(* CODESYS project CODESYS-Libraries
   Author: Ernesto Ponce
   Company: EPonce
   DefaultNamespace: SM_Control
   Description: This Library includes all FB, DUTs and Visualization Faceplates to use the State Machine Logic
   DocFormat: reStructuredText
   LanguageModelAttribute: qualified-access-only
   Placeholder: SM:
   Title: SM_Control
   Version: 1.0

Project tree, tasks and I/O mapping:
  libraries: Util, 3.5.19.0 (System); Standard, 3.5.18.0 (System); VisuSymbols, 4.4.0.0 (System); CmpBitmapPool, 3.5.17.0 (System); VisuDialogs, * (System)
  5ce3da45-db07-42e7-a21c-a00fff4ed8f6|Icons\abort_symbol.png
  5ce3da45-db07-42e7-a21c-a00fff4ed8f6|Icons\camera_icon.png
  5ce3da45-db07-42e7-a21c-a00fff4ed8f6|Icons\home_symbol.png
  5ce3da45-db07-42e7-a21c-a00fff4ed8f6|Icons\menu_icon.png
  5ce3da45-db07-42e7-a21c-a00fff4ed8f6|Icons\pause_symbol.png
  5ce3da45-db07-42e7-a21c-a00fff4ed8f6|Icons\permissives_icon.png
  5ce3da45-db07-42e7-a21c-a00fff4ed8f6|Icons\proceed_symbol.png
  5ce3da45-db07-42e7-a21c-a00fff4ed8f6|Icons\retry_symbol.png
  5ce3da45-db07-42e7-a21c-a00fff4ed8f6|Icons\start_symbol.png
  DUT/
    data type ActiveStep
    data type PermIntlkHMI_cfg
    data type PermIntlkHMI
    data type PermIntlkHMI_ocmd
    data type PermIntlkHMI_sts
    data type SM_HMI
    data type SM_HMI_cfg
    data type SM_HMI_ocmd
    data type SM_HMI_sts
  Function Blocks/
    function block Actuator [ST]: Advance, Reset_Faults, Retract
    function block Permissives [LD]
    program POU [LD]
    function block Real_From_Bytes [ST]
    function block StateMachine [LD]
    function block Step [LD]
  text list GlobalTextList
  global variables GVL
  image pool ImagePool
  Visu_Logic/
    program Visu_Logic [LD]
  Visualizations/
    visualisation Button
    visualisation Menu_Button
    visualisation Permissives_faceplate
    visualisation Screen_Navigation
    visualisation SM_faceplate
*)

// DUT/ActiveStep
TYPE ActiveStep  :
STRUCT
  Step : DINT;
  StatusStepFaulted : BOOL;
  PermsHMI : PermIntlkHMI;
END_STRUCT
END_TYPE

// DUT/PermIntlkHMI_cfg
TYPE PermIntlkHMI_cfg :
STRUCT
  Name : STRING;
  Desc : ARRAY [0..15] OF STRING;
END_STRUCT
END_TYPE

// DUT/PermIntlkHMI
TYPE PermIntlkHMI :
STRUCT
  cfg : PermIntlkHMI_cfg;
  ocmd : PermIntlkHMI_ocmd;
  sts : PermIntlkHMI_sts;
END_STRUCT
END_TYPE

// DUT/PermIntlkHMI_ocmd
TYPE PermIntlkHMI_ocmd :
STRUCT
  ForceOK : BOOL;
END_STRUCT
END_TYPE

// DUT/PermIntlkHMI_sts
TYPE PermIntlkHMI_sts :
STRUCT
  OK : BOOL;
  ForceOK : BOOL;
  PermIntlk : INT;
END_STRUCT
END_TYPE

// DUT/SM_HMI
TYPE SM_HMI :
STRUCT
  cfg : SM_HMI_cfg;
  ocmd : SM_HMI_ocmd;
  sts : SM_HMI_sts;
  NextStatePerms : PermIntlkHMI;
  ActiveStepHMI : PermIntlkHMI;
END_STRUCT
END_TYPE

// DUT/SM_HMI_cfg
TYPE SM_HMI_cfg :
STRUCT
  Name : STRING(40);
  HomePerm : PermIntlkHMI_cfg;
  StartPerm : PermIntlkHMI_cfg;
  ProceedPerm : PermIntlkHMI_cfg;
  AutoIntlk : PermIntlkHMI_cfg;
END_STRUCT
END_TYPE

// DUT/SM_HMI_ocmd
TYPE SM_HMI_ocmd :
STRUCT
  Abort : BOOL;
  Home : BOOL;
  Start : BOOL;
  Stop : BOOL;
  Pause : BOOL;
  Proceed : BOOL;
  Retry : BOOL;
  ActiveStatePermBypass : BOOL;
END_STRUCT
END_TYPE

// DUT/SM_HMI_sts
TYPE SM_HMI_sts :
STRUCT
  Automatic : BOOL;
  Manual : BOOL;
  StepMode : BOOL;
  Homing : BOOL;
  Homed : BOOL;
  Running : BOOL;
  Complete : BOOL;
  Stopping : BOOL;
  Stopped : BOOL;
  Aborting : BOOL;
  Aborted : BOOL;
  Pausing : BOOL;
  Paused : BOOL;
  Proceeding : BOOL;
  Faulted : BOOL;
  ChildFaulted : BOOL;
  ReadyToHome : BOOL;
  ReadyToProceed : BOOL;
  ReadyToStart : BOOL;
  AutoStartRequest : BOOL;
  AutoCycleRequest : BOOL;
  Blocked : BOOL;
  Starved : BOOL;
  Mode : DINT;
  Step : DINT;
  NextStep : DINT;
  ReturnNextStep : DINT;
END_STRUCT
END_TYPE

// GVL

VAR_GLOBAL
	// Global Variables for forcing values
	alwaysTrue : BOOL := TRUE;
	alwaysFalse : BOOL := FALSE;
	
	
	// Colors for Visualization
    indicatorRed: DWORD := 16#FF800000;    // Standard red color, fully opaque
    indicatorGreen: DWORD := 16#FF008000;  // Standard green color, fully opaque
    
    // Modern Color Palette for Buttons
    buttonRed: DWORD := 16#FFE57373;       // Rosy Red, opaque
    buttonRedDarker1: DWORD := 16#FFAF4448; // Crimson Red, opaque
    buttonRedDarker2: DWORD := 16#FF7B3034; // Dark Red, opaque
    buttonRedDarkest: DWORD := 16#FF541F21; // Maroon, opaque
    
    buttonGreen: DWORD := 16#FF81C784;     // Light Green, opaque
    buttonGreenDarker1: DWORD := 16#FF519657; // Medium Sea Green, opaque
    buttonGreenDarker2: DWORD := 16#FF346939; // Dark Green, opaque
    buttonGreenDarkest: DWORD := 16#FF234725; // Dark Olive Green, opaque
    
    buttonGrey: DWORD := 16#FFB0BEC5;      // Blue Grey, opaque
    buttonGreyDarker1: DWORD := 16#FF78909C; // Cadet Blue, opaque
    buttonGreyDarker2: DWORD := 16#FF546E7A; // Steel Blue, opaque
    buttonGreyDarkest: DWORD := 16#FF37474F; // Dark Slate Gray, opaque
	
	// Full Pallet Color Declaration
	
	// Green Palette
	GreenP_1: DWORD := 16#FF859191; // Lightest Green
	GreenP_2: DWORD := 16#FF6F8383; // Light Green
	GreenP_3: DWORD := 16#FF587474; // Medium Light Green
	GreenP_4: DWORD := 16#FF426666; // Medium Green
	GreenP_5: DWORD := 16#FF355151; // Medium Dark Green
	GreenP_6: DWORD := 16#FF283C3C; // Dark Green
	GreenP_7: DWORD := 16#FF1C2828; // Darkest Green
	
	// Grey Palette
	BlueP_1: DWORD := 16#FF8198AD; // Lightest Blue
	BlueP_2: DWORD := 16#FF718CA5; // Light Blue
	BlueP_3: DWORD := 16#FF61809D; // Medium Light Blue
	BlueP_4: DWORD := 16#FF517495; // Medium Blue
	BlueP_5: DWORD := 16#FF41617B; // Medium Dark Blue
	BlueP_6: DWORD := 16#FF314F60; // Dark Blue
	BlueP_7: DWORD := 16#FF213C46; // Darkest Blue
	
	// Purple Palette
	PurpleP_1: DWORD := 16#FF888ECC; // Lightest Purple
	PurpleP_2: DWORD := 16#FF8284C4; // Light Purple
	PurpleP_3: DWORD := 16#FF7C7BBC; // Medium Light Purple
	PurpleP_4: DWORD := 16#FF7571B4; // Medium Purple
	PurpleP_5: DWORD := 16#FF6F68AC; // Medium Dark Purple
	PurpleP_6: DWORD := 16#FF685EA4; // Dark Purple
	PurpleP_7: DWORD := 16#FF62549C; // Darkest Purple
	
	// Yellow Palette
	YellowP_1: DWORD := 16#FFCCC68C; // Lightest Yellow
	YellowP_2: DWORD := 16#FFC4BE80; // Light Yellow
	YellowP_3: DWORD := 16#FFBCB675; // Medium Light Yellow
	YellowP_4: DWORD := 16#FFB4AE6A; // Medium Yellow
	YellowP_5: DWORD := 16#FFACA65F; // Medium Dark Yellow
	YellowP_6: DWORD := 16#FFA49E54; // Dark Yellow
	YellowP_7: DWORD := 16#FF9C9648; // Darkest Yellow
	
	// Brown Palette
	BrownP_1: DWORD := 16#FF99836D; // Lightest Brown
	BrownP_2: DWORD := 16#FF8D7761; // Light Brown
	BrownP_3: DWORD := 16#FF816B55; // Medium Light Brown
	BrownP_4: DWORD := 16#FF755F49; // Medium Brown
	BrownP_5: DWORD := 16#FF69533D; // Medium Dark Brown
	BrownP_6: DWORD := 16#FF5D4731; // Dark Brown
	BrownP_7: DWORD := 16#FF513B25; // Darkest Brown
	
	// Darkened Grey UI Palette
	GreyP_1: DWORD := 16#FFB8B8BC;  // Light Grey
	GreyP_2: DWORD := 16#FFA8A8AC;  // Slightly lighter Grey
	GreyP_3: DWORD := 16#FF98989C;  // Medium Light Grey
	GreyP_4: DWORD := 16#FF88888C;  // True Medium Grey
	GreyP_5: DWORD := 16#FF78787C;  // Medium Dark Grey
	GreyP_6: DWORD := 16#FF68686C;  // Darker Grey
	GreyP_7: DWORD := 16#FF58585C;  // Dark Grey
	
	
	// Visualization Colors Using Pallet
	hover_color : DWORD := BlueP_4;
	normal_color : DWORD := BlueP_6;
	click_color : DWORD := BlueP_6;
	mouseDown_color : DWORD := BlueP_3;
	
	led_colorOFF : DWORD := GreenP_6;
	led_colorON : DWORD := GreenP_3;

END_VAR

// Function Blocks/Actuator
FUNCTION_BLOCK Actuator
VAR_INPUT
	EN:BOOL;
    inRetPermissive: Permissives;
    inAdvPermissive: Permissives;
    inAdvFeedback: BOOL;
    inRetFeedback: BOOL;
    cfgAdvTimeout: TIME;
    cfgRetTimeout: TIME;
END_VAR

VAR_OUTPUT
	ENOut:BOOL;
    outAdvance: BOOL;
    outRetract: BOOL;
	stsAdvancing: BOOL;
    stsAdvanced: BOOL;
	stsRetracting: BOOL;
    stsRetracted: BOOL;
    stsFaulted: BOOL;
    stsFaultCode: INT;
END_VAR

VAR_IN_OUT
	HMI: PermIntlkHMI;
END_VAR


VAR
	timeAdvance:TON;
	timeRetract:TON;	
END_VAR

stsAdvanced:=inAdvFeedback;
stsRetracted:=inRetFeedback;

inAdvPermissive(HMI := HMI);
inRetPermissive(HMI := HMI);


(*
Timeout Fault
Faulted Reason Codes:

- stsFaultCode.0 = 1 = Requested to Advance but !PermsOK
- stsFaultCode.1 = 2 = Requested to Retract but !PermsOK
- stsFaultCode.2 = 4 = Interlocks are not OK
- stsFaultCode.3 = 8 = Advance Timeout
- stsFaultCode.4 = 16 = Retract Timeout
*)
	
timeAdvance(IN:= outAdvance, PT:=cfgAdvTimeout);	
	
IF stsAdvancing AND timeAdvance.Q AND  NOT(inAdvFeedback) THEN
	outAdvance := 0;
	outRetract := 0;
	stsRetracting := 0;
	stsAdvancing := 0;
	stsFaulted := 1;
	stsFaultCode := 8;
END_IF

timeRetract(IN:= outRetract, PT:=cfgRetTimeout);

IF stsRetracting AND timeRetract.Q  AND  NOT(inRetFeedback)THEN
	outAdvance := 0;
	outRetract := 0;
	stsRetracting := 0;
	stsAdvancing := 0;
	stsFaulted := 1;
	stsFaultCode := 16;
END_IF

IF outAdvance AND stsAdvanced THEN	
	stsAdvancing := 0;
END_IF

IF outRetract AND stsRetracted THEN	
	stsRetracting := 0;
END_IF

METHOD Advance : BOOL
VAR_INPUT
	pcmdAdvance:BOOL;
	
END_VAR

VAR
	ONS : R_TRIG;
	
	test:BOOL;
END_VAR
// Advance Logic
ONS(clk:=pcmdAdvance);

IF ONS.Q AND NOT(stsretracting OR stsAdvancing) THEN
	
	outRetract := 0;

	
	IF inAdvPermissive.stsOk THEN
		outAdvance := 1;
		stsAdvancing:= 1;		
	ELSE
		outAdvance := 0;
		outRetract := 0;		
		stsFaulted := 1;
		stsFaultCode := 1;
	END_IF
		
	
END_IF
END_METHOD

METHOD Reset_Faults : BOOL
VAR_INPUT
	pcmdResetFaults:BOOL;
	
END_VAR

VAR
	ONS : R_TRIG;
	
	test:BOOL;
END_VAR
ONS(clk:=pcmdResetFaults);

IF ONS.Q THEN
	outAdvance := 0;
	outRetract := 0;
	stsFaulted := 0;
	stsFaultCode := 0;	
END_IF
END_METHOD

METHOD Retract : BOOL
VAR_INPUT
	pcmdRetract:BOOL;
	
END_VAR

VAR
	ONS : R_TRIG;
	
END_VAR
// Retract Logic
ONS(clk:=pcmdRetract);

IF ONS.Q AND NOT(stsretracting OR stsAdvancing)THEN
	
	outAdvance := 0;

	
	IF inAdvPermissive.stsOk THEN
		outRetract := 1;
		stsRetracting := 1;		
	ELSE
		outAdvance := 0;
		outRetract := 0;
		stsFaulted := 1;
		stsFaultCode := 2;
	END_IF
	
	
END_IF
END_METHOD

END_FUNCTION_BLOCK

// Function Blocks/Permissives
FUNCTION_BLOCK Permissives
VAR_INPUT
	EN: BOOL;
	inPermissives: int;
	ocmdForceOk: BOOL;
	
END_VAR
VAR_OUTPUT
	ENOut: BOOL;
	stsOk: BOOL;
	stsForceOk: BOOL;
	
END_VAR
VAR
END_VAR

VAR_IN_OUT
	HMI: PermIntlkHMI;
END_VAR
VAR // added by the converter: edge detectors and wires of the graphical bodies
    _w1, _w2 : BOOL;
END_VAR

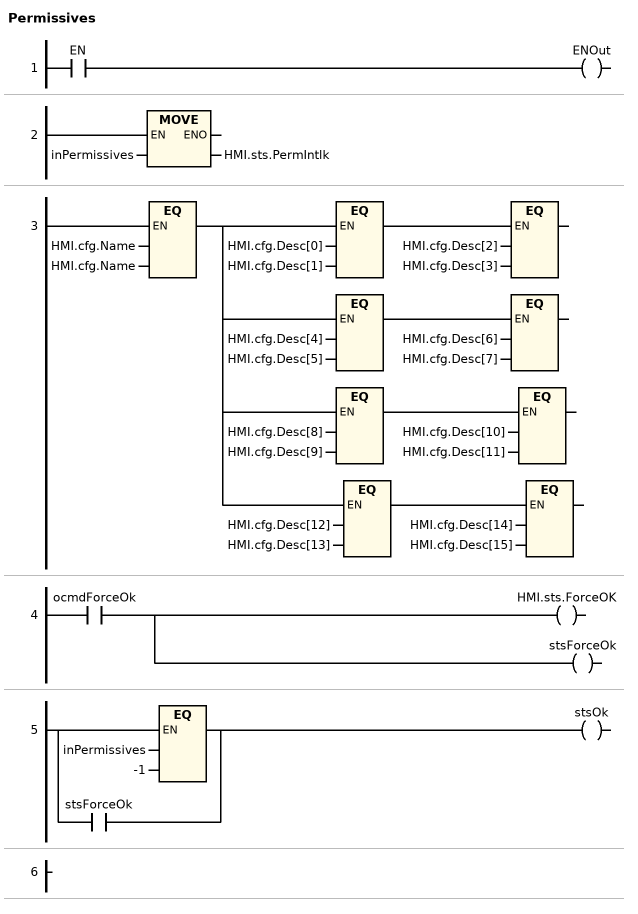
// NETWORK 1
ENOut := EN;

// NETWORK 2
HMI.sts.PermIntlk := inPermissives;

// NETWORK 3
_w1 := HMI.cfg.Name = HMI.cfg.Name;
(* _w1 AND HMI.cfg.Desc[0] = HMI.cfg.Desc[1] AND HMI.cfg.Desc[2] = HMI.cfg.Desc[3]; result not used *)
(* _w1 AND HMI.cfg.Desc[4] = HMI.cfg.Desc[5] AND HMI.cfg.Desc[6] = HMI.cfg.Desc[7]; result not used *)
(* _w1 AND HMI.cfg.Desc[8] = HMI.cfg.Desc[9] AND HMI.cfg.Desc[10] = HMI.cfg.Desc[11]; result not used *)
(* _w1 AND HMI.cfg.Desc[12] = HMI.cfg.Desc[13] AND HMI.cfg.Desc[14] = HMI.cfg.Desc[15]; result not used *)

// NETWORK 4
HMI.sts.ForceOK := ocmdForceOk;
stsForceOk := ocmdForceOk;

// NETWORK 5
_w2 := stsForceOk;
IF NOT _w2 THEN
    _w2 := inPermissives = -1;
END_IF
stsOk := _w2;

// NETWORK 6

END_FUNCTION_BLOCK

// Function Blocks/POU
PROGRAM POU
VAR
	
END_VAR

// NETWORK 1

END_PROGRAM

// Function Blocks/Real_From_Bytes
FUNCTION_BLOCK Real_From_Bytes
VAR_INPUT
    Byte1: BYTE; 
    Byte2: BYTE; 
    Byte3: BYTE; 
    Byte4: BYTE; 
END_VAR

VAR_OUTPUT
    RealValue: REAL; // The resulting REAL value
    
END_VAR

VAR
    Word1: WORD;
    Word2: WORD;
    Word3: WORD;
    Word4: WORD;
    Dword1: DWORD;
    Dword2: DWORD;
    Dword3: DWORD;
    Dword4: DWORD;
    ShiftedDword2: DWORD;
    ShiftedDword3: DWORD;
    ShiftedDword4: DWORD;
	CombinedDword: DWORD;
    ptrRealValue: POINTER TO REAL;
END_VAR

 // Convert each byte to a WORD
    Word1 := BYTE_TO_WORD(Byte4);
    Word2 := BYTE_TO_WORD(Byte1);
    Word3 := BYTE_TO_WORD(Byte2);
    Word4 := BYTE_TO_WORD(Byte3);

    // Convert each WORD to a DWORD
    Dword1 := WORD_TO_DWORD(Word1);
    Dword2 := WORD_TO_DWORD(Word2);
    Dword3 := WORD_TO_DWORD(Word3);
    Dword4 := WORD_TO_DWORD(Word4);

    // Shift DWORDs to the correct position
    ShiftedDword2 := SHL(Dword2, 8);
    ShiftedDword3 := SHL(Dword3, 16);
    ShiftedDword4 := SHL(Dword4, 24);

    // Combine the DWORDs into one DWORD assuming big-endian order
    CombinedDword := Dword1 OR ShiftedDword2 OR ShiftedDword3 OR ShiftedDword4;

    // Use pointer method to convert the combined DWORD to REAL
    ptrRealValue := ADR(CombinedDword);
    RealValue := ptrRealValue^;

END_FUNCTION_BLOCK

// Function Blocks/StateMachine
FUNCTION_BLOCK StateMachine

VAR_INPUT
    EnableIn: BOOL;
    cfgAutoRun: BOOL;
    inpAutoIntlk: INT:= -1;
    inpBlockedCondition: DINT;
    inpHomePerm: INT := -1;
    inpProceedPerm: INT := -1;
    inpStartPerm: INT := -1;
    inpStarvedCondition: DINT;
    inpSubmoduleFaulted: BOOL;
    NextStep: DINT;
    pcmdAbort: BOOL;
    pcmdCompleteState: BOOL;
    pcmdHome: BOOL;
    pcmdPause: BOOL;
    pcmdProceed: BOOL;
    pcmdRetry: BOOL;
    pcmdStart: BOOL;
    pcmdStop: BOOL;
END_VAR

VAR_OUTPUT
    EnableOut: BOOL;
    outRetry: BOOL;
    stsAborted: BOOL;
    stsAborting: BOOL;
    stsActiveState: BOOL;
    stsAutoCycleRequest: BOOL;
    stsAutoIntlkOK: BOOL;
    stsAutomatic: BOOL;
    stsAutoStartRequest: BOOL;
    stsBlocked: BOOL;
    stsBlockedCondition: DINT;
    stsComplete: BOOL;
    stsFaulted: BOOL;
    stsHomed: BOOL;
    stsHomePermOk: BOOL;
    stsHoming: BOOL;
    stsManual: BOOL;
    stsMode: DINT;
    stsPaused: BOOL;
    stsPausing: BOOL;
    stsProceeding: BOOL;
    stsProceedPermOK: BOOL;
    stsReadyToHome: BOOL;
    stsReadyToProceed: BOOL;
    stsReadyToStart: BOOL;
    stsReturnNextStep: DINT;
    stsRunning: BOOL;
    stsStartPermOK: BOOL;
    stsStarved: BOOL;
    stsStarvedCondition: DINT;
    stsStep: DINT;
    stsStepTimerSeconds: REAL;
    stsStopped: BOOL;
    stsStopping: BOOL;
    stsSubmoduleFaulted: BOOL;
    stsWaitingState: BOOL;
	stsState: INT;
	stsStateString: STRING;
	stsReturnState: INT;
	stsLastState: INT;
END_VAR


VAR CONSTANT 
	internalClearStep: ActiveStep;  
	EmptyHMIPerm: PermIntlkHMI;
	
	// All internal steps
	internalStateRunning: INT := 1;
    internalStateStopping: INT := 2;
    internalStateHoming: INT := 4;
    internalStateAborting: INT := 8;
    internalStateHomed: INT := 16;
    internalStateStopped: INT := 32;
    internalStateAborted: INT := 64;
    internalStateComplete: INT := 128;
    internalStatePausing: INT := 256;
    internalStatePaused: INT := 512;
    internalStateProceeding: INT := 1024;
END_VAR

VAR
    AbortRequested: BOOL;
    AutoStartRequested: BOOL;
    CompleteStateRequested: BOOL;
    HomeRequested: BOOL;
    PauseRequested: BOOL;
    ProceedRequested: BOOL;
    RetryComplete: BOOL;
    RetryRequested: BOOL;
    StartRequested: BOOL;
    StopRequested: BOOL;
    StepTimer: TON;

    internalLsOdd: DINT;
   	internalONS: DINT;
 	R_TRIG_0: R_TRIG;
	R_TRIG_1: R_TRIG;
	R_TRIG_2: R_TRIG;
	R_TRIG_3: R_TRIG;
	internalTimerReset: BOOL;
	
	internalPauseStep: ActiveStep;
    internalPreviousState: INT;
	internalAutoIntlk: Permissives;
    internalAutoIntlk_HMI: PermIntlkHMI;
    internalProceedPerm: Permissives;
    internalProceedPerm_HMI: PermIntlkHMI;
    internalStartPerm: Permissives;
    internalStartPerm_HMI: PermIntlkHMI;
	internalHomePerm: Permissives;
    internalHomePerm_HMI: PermIntlkHMI;
	internalStepHistoryMax: DINT;
END_VAR


VAR_IN_OUT 
    HMI: SM_HMI;
    CurrentStep: ActiveStep;
    
END_VAR
VAR // added by the converter: edge detectors and wires of the graphical bodies
    _w1, _w2, _w3, _w4, _w5, _w6, _w7, _w8, _w9, _w10, _w11, _w12, _w13, _w14, _w15, _w16, _w17, _w18, _w19, _w20, _w21, _w22, _w23, _w24, _w25, _w26, _w27, _w28, _w29, _w30, _w31, _w32, _w33, _w34, _w35, _w36, _w37, _w38, _w39, _w40, _w41, _w42, _w43, _w44 : BOOL;
    _rt1, _rt2 : R_TRIG;
END_VAR

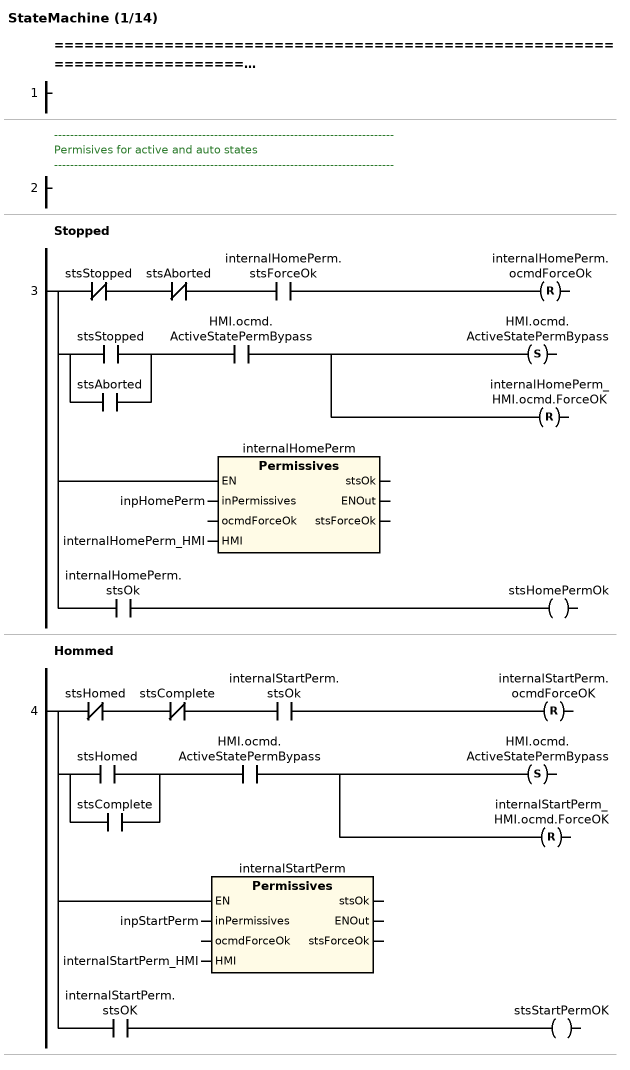
// NETWORK 1: ============================================================================ State Machine ============================================================================ (disabled)

// NETWORK 2
// -------------------------------------------------------------------------------------
//
// Permisives for active and auto states
//
// -------------------------------------------------------------------------------------

// NETWORK 3: Stopped
internalHomePerm.ocmdForceOk R= NOT stsStopped AND NOT stsAborted AND internalHomePerm.stsForceOk;
_w1 := (stsStopped OR stsAborted) AND HMI.ocmd.ActiveStatePermBypass;
HMI.ocmd.ActiveStatePermBypass S= _w1;
internalHomePerm_HMI.ocmd.ForceOK R= _w1;
internalHomePerm(EN := TRUE, inPermissives := inpHomePerm, HMI := internalHomePerm_HMI); // Permissives
stsHomePermOk := internalHomePerm.stsOk;

// NETWORK 4: Hommed
internalStartPerm.ocmdForceOK R= NOT stsHomed AND NOT stsComplete AND internalStartPerm.stsOk;
_w2 := (stsHomed OR stsComplete) AND HMI.ocmd.ActiveStatePermBypass;
HMI.ocmd.ActiveStatePermBypass S= _w2;
internalStartPerm_HMI.ocmd.ForceOK R= _w2;
internalStartPerm(EN := TRUE, inPermissives := inpStartPerm, HMI := internalStartPerm_HMI); // Permissives
stsStartPermOK := internalStartPerm.stsOK;

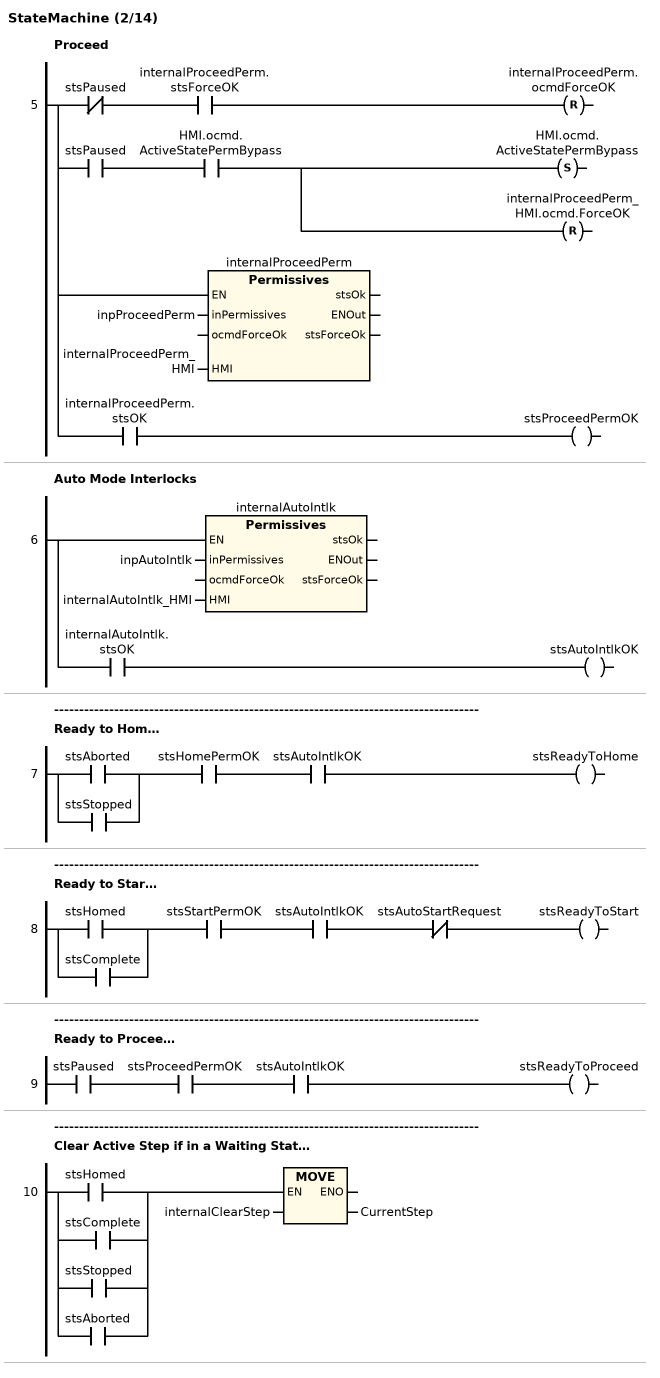
// NETWORK 5: Proceed
internalProceedPerm.ocmdForceOK R= NOT stsPaused AND internalProceedPerm.stsForceOK;
_w3 := stsPaused AND HMI.ocmd.ActiveStatePermBypass;
HMI.ocmd.ActiveStatePermBypass S= _w3;
internalProceedPerm_HMI.ocmd.ForceOK R= _w3;
internalProceedPerm(EN := TRUE, inPermissives := inpProceedPerm, HMI := internalProceedPerm_HMI); // Permissives
stsProceedPermOK := internalProceedPerm.stsOK;

// NETWORK 6: Auto Mode Interlocks
internalAutoIntlk(EN := TRUE, inPermissives := inpAutoIntlk, HMI := internalAutoIntlk_HMI); // Permissives
stsAutoIntlkOK := internalAutoIntlk.stsOK;

// NETWORK 7: ------------------------------------------------------------------------------------- Ready to Home - if stopped or aborted - if Perms are OK -------------------------------------------------------------------------------------
stsReadyToHome := (stsAborted OR stsStopped) AND stsHomePermOK AND stsAutoIntlkOK;

// NETWORK 8: ------------------------------------------------------------------------------------- Ready to Start - if homed or complete - if Perms are OK -------------------------------------------------------------------------------------
stsReadyToStart := (stsHomed OR stsComplete) AND stsStartPermOK AND stsAutoIntlkOK AND NOT stsAutoStartRequest;

// NETWORK 9: ------------------------------------------------------------------------------------- Ready to Proceed - if paused - if Perms are OK -------------------------------------------------------------------------------------
stsReadyToProceed := stsPaused AND stsProceedPermOK AND stsAutoIntlkOK;

// NETWORK 10: ------------------------------------------------------------------------------------- Clear Active Step if in a Waiting State -------------------------------------------------------------------------------------
IF stsHomed OR stsComplete OR stsStopped OR stsAborted THEN CurrentStep := internalClearStep; END_IF

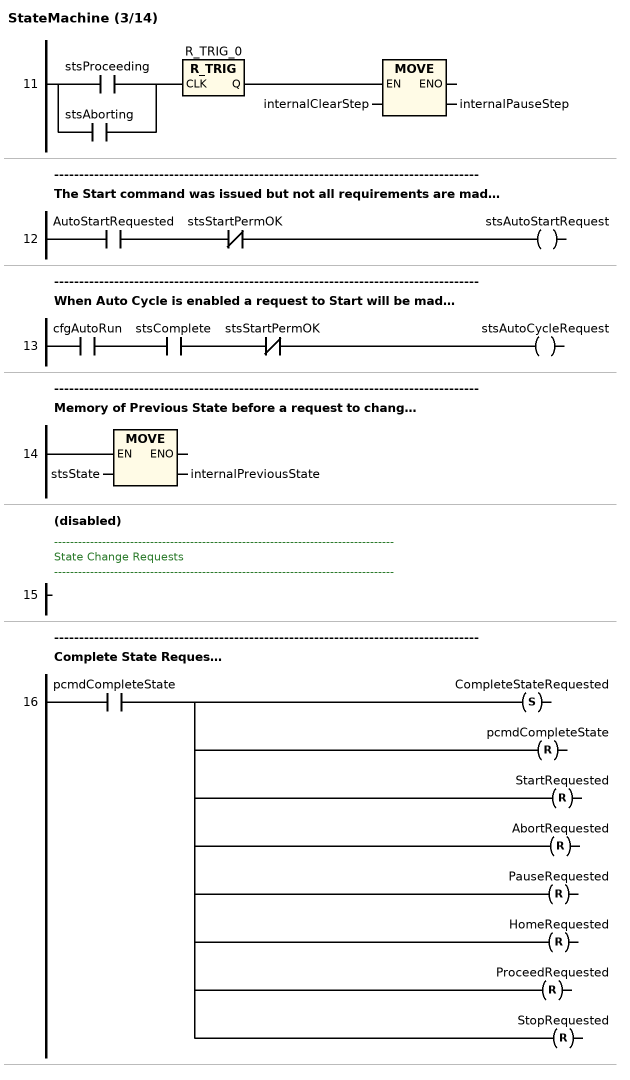
// NETWORK 11
R_TRIG_0(CLK := stsProceeding OR stsAborting); // R_TRIG
IF R_TRIG_0.Q THEN internalPauseStep := internalClearStep; END_IF

// NETWORK 12: ------------------------------------------------------------------------------------- The Start command was issued but not all requirements are made The request will be remembered and this will happen as soon as everything is ready to Start -------------------------------------------------------------------------------------
stsAutoStartRequest := AutoStartRequested AND NOT stsStartPermOK;

// NETWORK 13: ------------------------------------------------------------------------------------- When Auto Cycle is enabled a request to Start will be made as soon as the previous cycle is Complete -------------------------------------------------------------------------------------
stsAutoCycleRequest := cfgAutoRun AND stsComplete AND NOT stsStartPermOK;

// NETWORK 14: ------------------------------------------------------------------------------------- Memory of Previous State before a request to change -------------------------------------------------------------------------------------
internalPreviousState := stsState;

// NETWORK 15 (disabled)
// -------------------------------------------------------------------------------------
//
// State Change Requests
//
// -------------------------------------------------------------------------------------

// NETWORK 16: ------------------------------------------------------------------------------------- Complete State Request -------------------------------------------------------------------------------------
_w4 := pcmdCompleteState;
CompleteStateRequested S= _w4;
pcmdCompleteState R= _w4;
StartRequested R= _w4;
AbortRequested R= _w4;
PauseRequested R= _w4;
HomeRequested R= _w4;
ProceedRequested R= _w4;
StopRequested R= _w4;

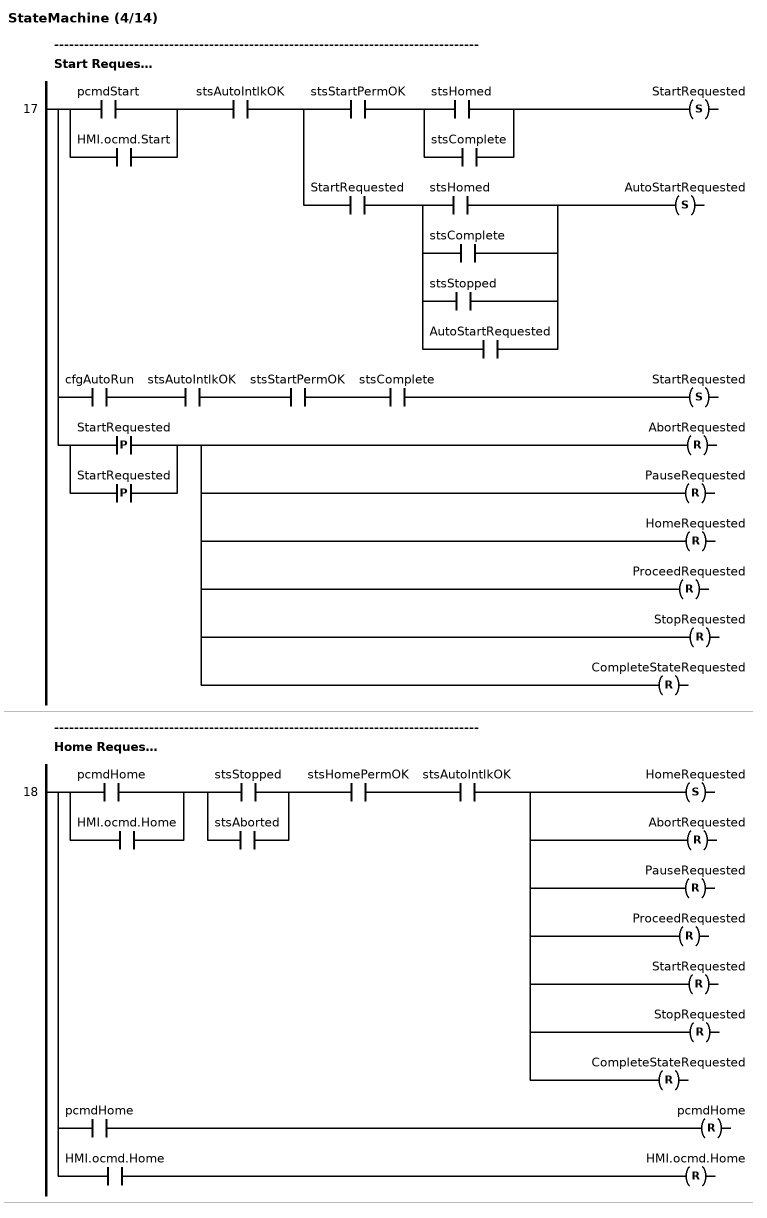
// NETWORK 17: ------------------------------------------------------------------------------------- Start Request -------------------------------------------------------------------------------------
_w5 := (pcmdStart OR HMI.ocmd.Start) AND stsAutoIntlkOK;
StartRequested S= _w5 AND stsStartPermOK AND (stsHomed OR stsComplete);
AutoStartRequested S= _w5 AND StartRequested AND (stsHomed OR stsComplete OR stsStopped OR AutoStartRequested);
StartRequested S= cfgAutoRun AND stsAutoIntlkOK AND stsStartPermOK AND stsComplete;
_rt1(CLK := StartRequested);
_rt2(CLK := StartRequested);
_w6 := _rt1.Q OR _rt2.Q;
AbortRequested R= _w6;
PauseRequested R= _w6;
HomeRequested R= _w6;
ProceedRequested R= _w6;
StopRequested R= _w6;
CompleteStateRequested R= _w6;

// NETWORK 18: ------------------------------------------------------------------------------------- Home Request -------------------------------------------------------------------------------------
_w7 := (pcmdHome OR HMI.ocmd.Home) AND (stsStopped OR stsAborted) AND stsHomePermOK AND stsAutoIntlkOK;
HomeRequested S= _w7;
AbortRequested R= _w7;
PauseRequested R= _w7;
ProceedRequested R= _w7;
StartRequested R= _w7;
StopRequested R= _w7;
CompleteStateRequested R= _w7;
pcmdHome R= pcmdHome;
HMI.ocmd.Home R= HMI.ocmd.Home;

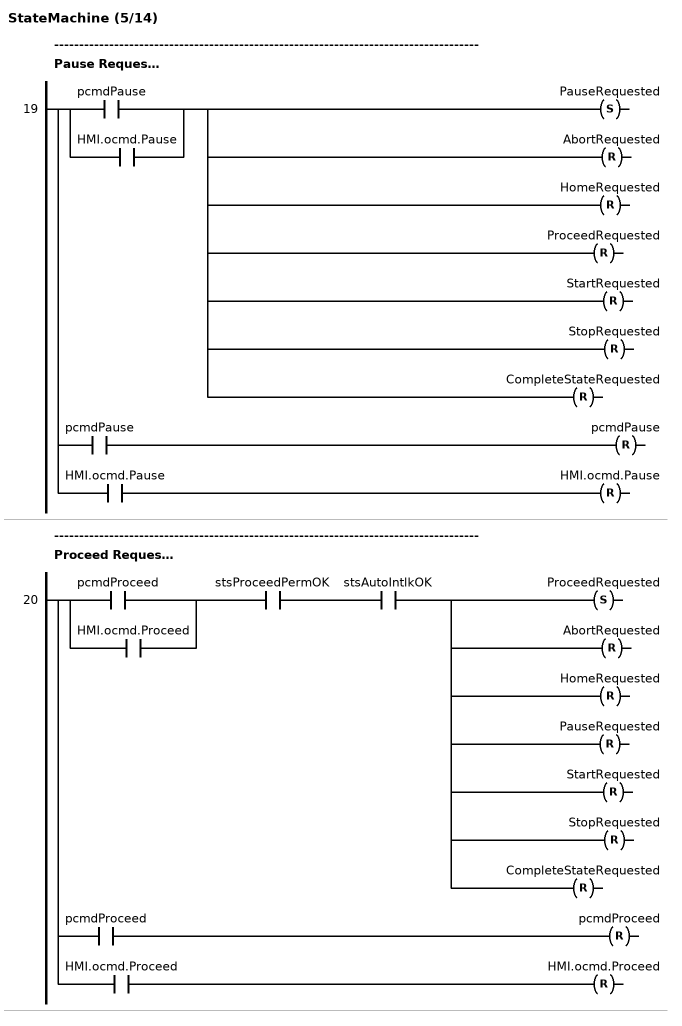
// NETWORK 19: ------------------------------------------------------------------------------------- Pause Request -------------------------------------------------------------------------------------
_w8 := pcmdPause OR HMI.ocmd.Pause;
PauseRequested S= _w8;
AbortRequested R= _w8;
HomeRequested R= _w8;
ProceedRequested R= _w8;
StartRequested R= _w8;
StopRequested R= _w8;
CompleteStateRequested R= _w8;
pcmdPause R= pcmdPause;
HMI.ocmd.Pause R= HMI.ocmd.Pause;

// NETWORK 20: ------------------------------------------------------------------------------------- Proceed Request -------------------------------------------------------------------------------------
_w9 := (pcmdProceed OR HMI.ocmd.Proceed) AND stsProceedPermOK AND stsAutoIntlkOK;
ProceedRequested S= _w9;
AbortRequested R= _w9;
HomeRequested R= _w9;
PauseRequested R= _w9;
StartRequested R= _w9;
StopRequested R= _w9;
CompleteStateRequested R= _w9;
pcmdProceed R= pcmdProceed;
HMI.ocmd.Proceed R= HMI.ocmd.Proceed;

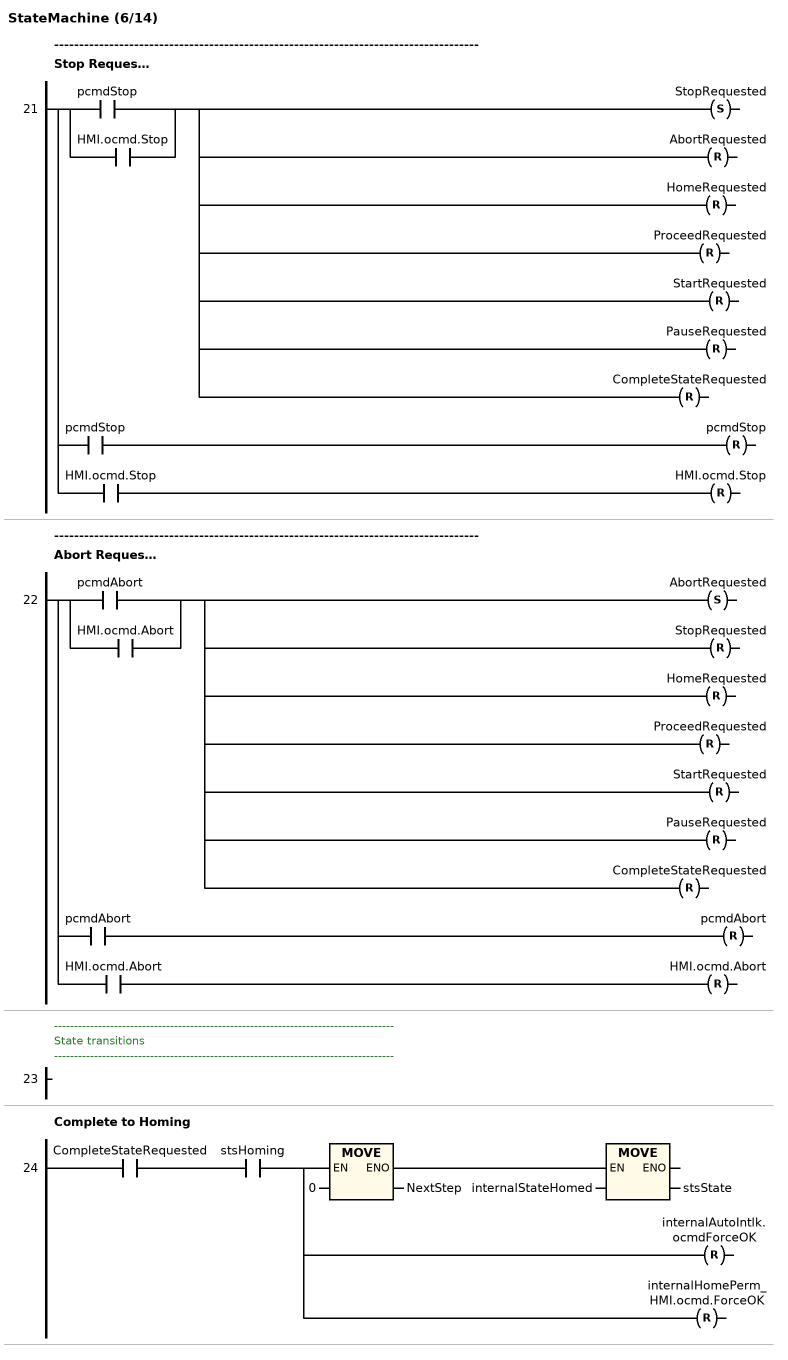
// NETWORK 21: ------------------------------------------------------------------------------------- Stop Request -------------------------------------------------------------------------------------
_w10 := pcmdStop OR HMI.ocmd.Stop;
StopRequested S= _w10;
AbortRequested R= _w10;
HomeRequested R= _w10;
ProceedRequested R= _w10;
StartRequested R= _w10;
PauseRequested R= _w10;
CompleteStateRequested R= _w10;
pcmdStop R= pcmdStop;
HMI.ocmd.Stop R= HMI.ocmd.Stop;

// NETWORK 22: ------------------------------------------------------------------------------------- Abort Request -------------------------------------------------------------------------------------
_w11 := pcmdAbort OR HMI.ocmd.Abort;
AbortRequested S= _w11;
StopRequested R= _w11;
HomeRequested R= _w11;
ProceedRequested R= _w11;
StartRequested R= _w11;
PauseRequested R= _w11;
CompleteStateRequested R= _w11;
pcmdAbort R= pcmdAbort;
HMI.ocmd.Abort R= HMI.ocmd.Abort;

// NETWORK 23
// -------------------------------------------------------------------------------------
//
// State transitions
//
// -------------------------------------------------------------------------------------

// NETWORK 24: Complete to Homing
_w12 := CompleteStateRequested AND stsHoming;
IF _w12 THEN NextStep := 0; END_IF
IF _w12 THEN stsState := internalStateHomed; END_IF
internalAutoIntlk.ocmdForceOK R= _w12;
internalHomePerm_HMI.ocmd.ForceOK R= _w12;

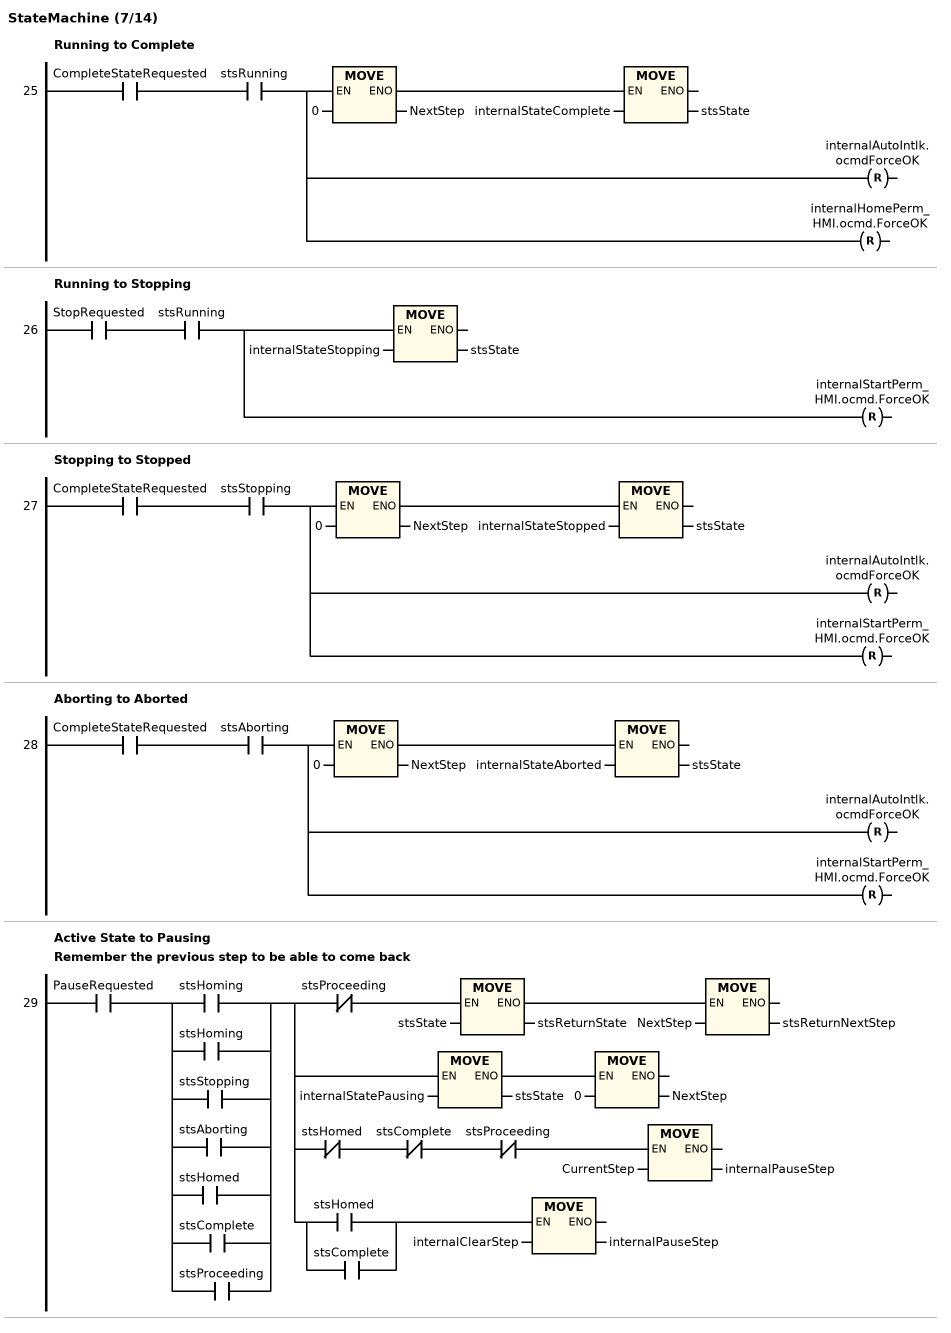
// NETWORK 25: Running to Complete
_w13 := CompleteStateRequested AND stsRunning;
IF _w13 THEN NextStep := 0; END_IF
IF _w13 THEN stsState := internalStateComplete; END_IF
internalAutoIntlk.ocmdForceOK R= _w13;
internalHomePerm_HMI.ocmd.ForceOK R= _w13;

// NETWORK 26: Running to Stopping
_w14 := StopRequested AND stsRunning;
IF _w14 THEN stsState := internalStateStopping; END_IF
internalStartPerm_HMI.ocmd.ForceOK R= _w14;

// NETWORK 27: Stopping to Stopped
_w15 := CompleteStateRequested AND stsStopping;
IF _w15 THEN NextStep := 0; END_IF
IF _w15 THEN stsState := internalStateStopped; END_IF
internalAutoIntlk.ocmdForceOK R= _w15;
internalStartPerm_HMI.ocmd.ForceOK R= _w15;

// NETWORK 28: Aborting to Aborted
_w16 := CompleteStateRequested AND stsAborting;
IF _w16 THEN NextStep := 0; END_IF
IF _w16 THEN stsState := internalStateAborted; END_IF
internalAutoIntlk.ocmdForceOK R= _w16;
internalStartPerm_HMI.ocmd.ForceOK R= _w16;

// NETWORK 29: Active State to Pausing Remember the previous step to be able to come back
_w17 := PauseRequested AND (stsHoming OR stsHoming OR stsStopping OR stsAborting OR stsHomed OR stsComplete OR stsProceeding);
IF _w17 AND NOT stsProceeding THEN stsReturnState := stsState; END_IF
IF _w17 AND NOT stsProceeding THEN stsReturnNextStep := NextStep; END_IF
IF _w17 THEN stsState := internalStatePausing; END_IF
IF _w17 THEN NextStep := 0; END_IF
IF _w17 AND NOT stsHomed AND NOT stsComplete AND NOT stsProceeding THEN internalPauseStep := CurrentStep; END_IF
IF _w17 AND (stsHomed OR stsComplete) THEN internalPauseStep := internalClearStep; END_IF

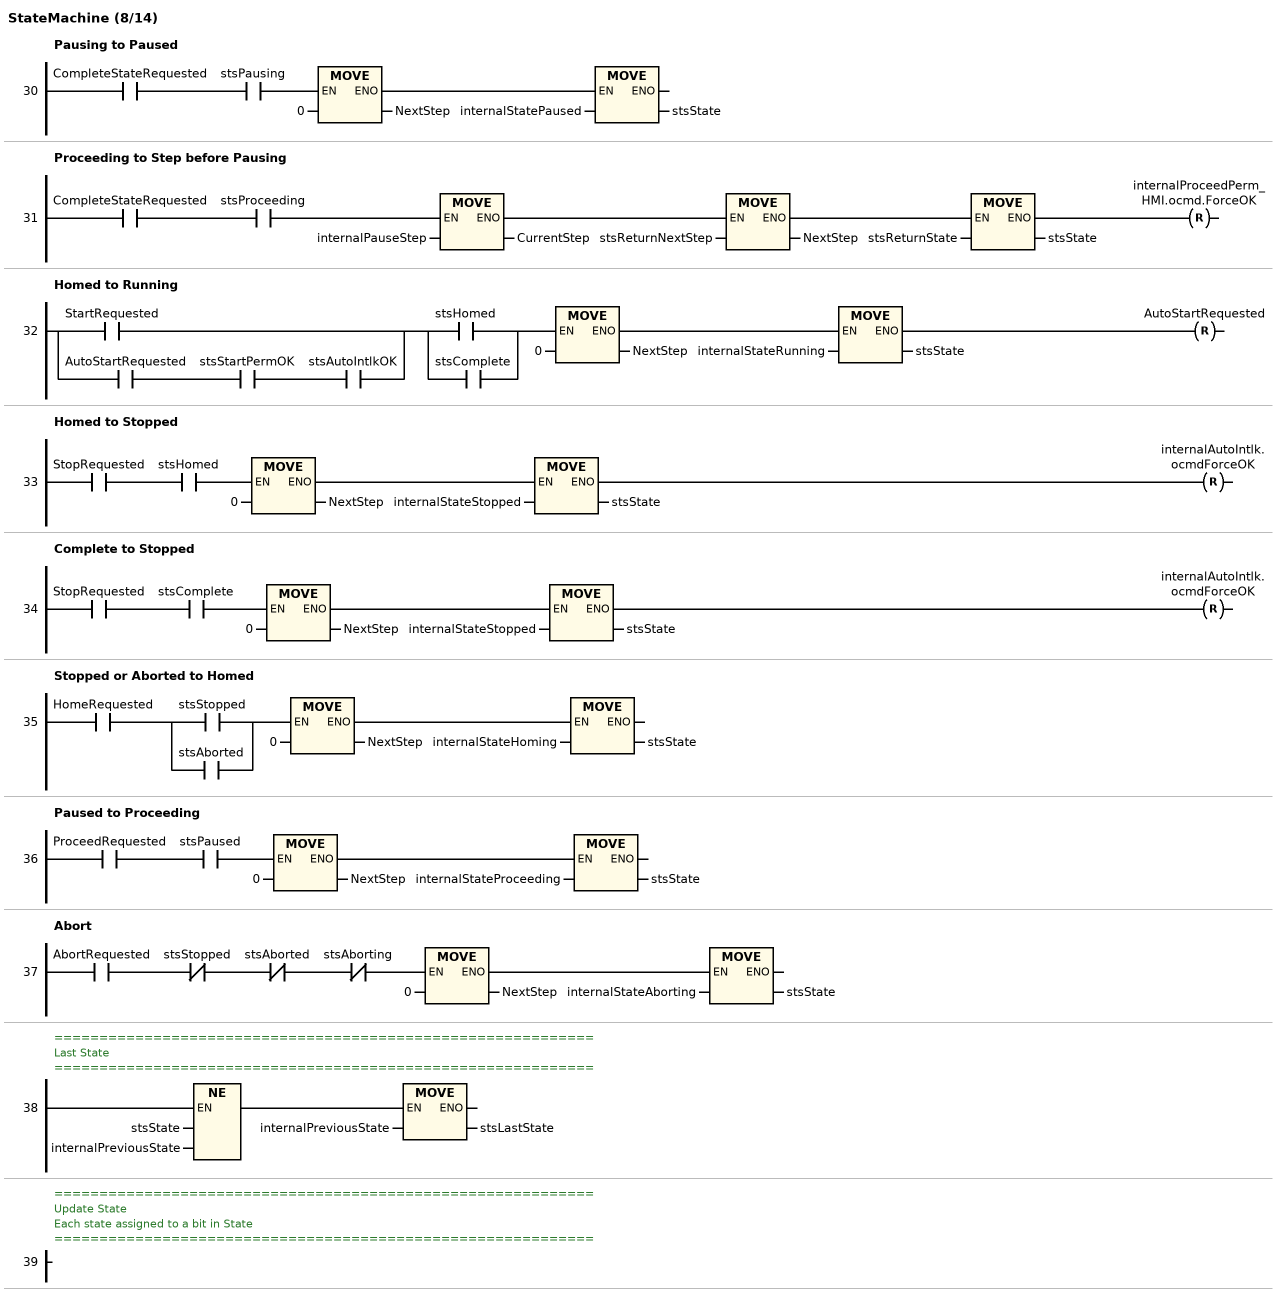
// NETWORK 30: Pausing to Paused
_w18 := CompleteStateRequested AND stsPausing;
IF _w18 THEN NextStep := 0; END_IF
IF _w18 THEN stsState := internalStatePaused; END_IF

// NETWORK 31: Proceeding to Step before Pausing
_w19 := CompleteStateRequested AND stsProceeding;
IF _w19 THEN CurrentStep := internalPauseStep; END_IF
IF _w19 THEN NextStep := stsReturnNextStep; END_IF
IF _w19 THEN stsState := stsReturnState; END_IF
internalProceedPerm_HMI.ocmd.ForceOK R= _w19;

// NETWORK 32: Homed to Running
_w20 := (StartRequested OR AutoStartRequested AND stsStartPermOK AND stsAutoIntlkOK) AND (stsHomed OR stsComplete);
IF _w20 THEN NextStep := 0; END_IF
IF _w20 THEN stsState := internalStateRunning; END_IF
AutoStartRequested R= _w20;

// NETWORK 33: Homed to Stopped
_w21 := StopRequested AND stsHomed;
IF _w21 THEN NextStep := 0; END_IF
IF _w21 THEN stsState := internalStateStopped; END_IF
internalAutoIntlk.ocmdForceOK R= _w21;

// NETWORK 34: Complete to Stopped
_w22 := StopRequested AND stsComplete;
IF _w22 THEN NextStep := 0; END_IF
IF _w22 THEN stsState := internalStateStopped; END_IF
internalAutoIntlk.ocmdForceOK R= _w22;

// NETWORK 35: Stopped or Aborted to Homed
_w23 := HomeRequested AND (stsStopped OR stsAborted);
IF _w23 THEN NextStep := 0; END_IF
IF _w23 THEN stsState := internalStateHoming; END_IF

// NETWORK 36: Paused to Proceeding
_w24 := ProceedRequested AND stsPaused;
IF _w24 THEN NextStep := 0; END_IF
IF _w24 THEN stsState := internalStateProceeding; END_IF

// NETWORK 37: Abort
_w25 := AbortRequested AND NOT stsStopped AND NOT stsAborted AND NOT stsAborting;
IF _w25 THEN NextStep := 0; END_IF
IF _w25 THEN stsState := internalStateAborting; END_IF

// NETWORK 38
// ============================================================
// Last State
// ============================================================
IF stsState <> internalPreviousState THEN stsLastState := internalPreviousState; END_IF

// NETWORK 39
// ============================================================
// Update State
// Each state assigned to a bit in State
// ============================================================

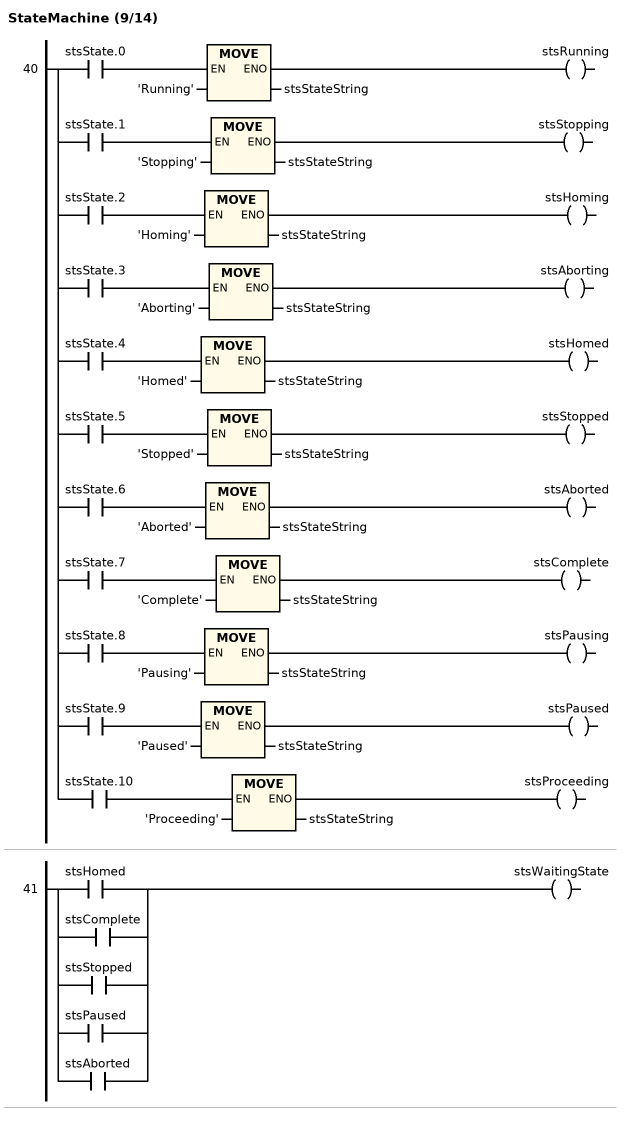
// NETWORK 40
_w26 := stsState.0;
IF _w26 THEN stsStateString := 'Running'; END_IF
stsRunning := _w26;
_w27 := stsState.1;
IF _w27 THEN stsStateString := 'Stopping'; END_IF
stsStopping := _w27;
_w28 := stsState.2;
IF _w28 THEN stsStateString := 'Homing'; END_IF
stsHoming := _w28;
_w29 := stsState.3;
IF _w29 THEN stsStateString := 'Aborting'; END_IF
stsAborting := _w29;
_w30 := stsState.4;
IF _w30 THEN stsStateString := 'Homed'; END_IF
stsHomed := _w30;
_w31 := stsState.5;
IF _w31 THEN stsStateString := 'Stopped'; END_IF
stsStopped := _w31;
_w32 := stsState.6;
IF _w32 THEN stsStateString := 'Aborted'; END_IF
stsAborted := _w32;
_w33 := stsState.7;
IF _w33 THEN stsStateString := 'Complete'; END_IF
stsComplete := _w33;
_w34 := stsState.8;
IF _w34 THEN stsStateString := 'Pausing'; END_IF
stsPausing := _w34;
_w35 := stsState.9;
IF _w35 THEN stsStateString := 'Paused'; END_IF
stsPaused := _w35;
_w36 := stsState.10;
IF _w36 THEN stsStateString := 'Proceeding'; END_IF
stsProceeding := _w36;

// NETWORK 41
stsWaitingState := stsHomed OR stsComplete OR stsStopped OR stsPaused OR stsAborted;

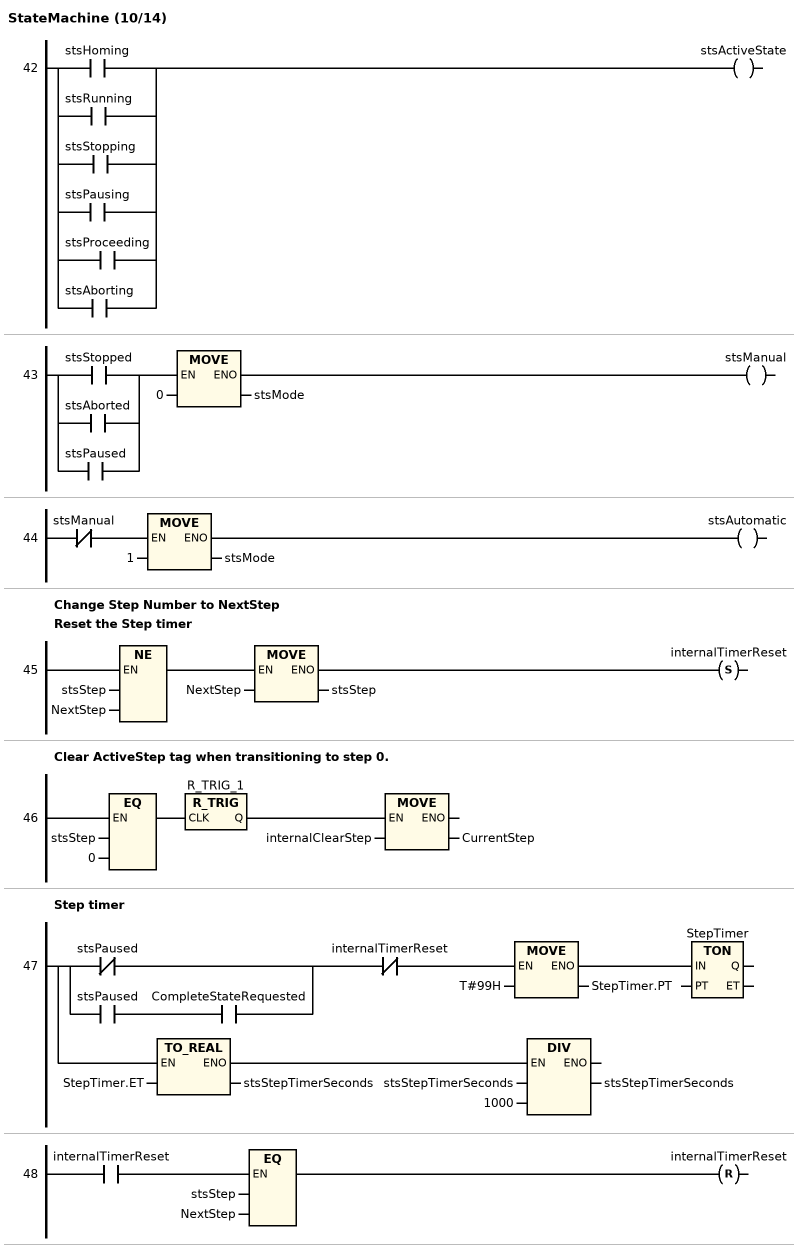
// NETWORK 42
stsActiveState := stsHoming OR stsRunning OR stsStopping OR stsPausing OR stsProceeding OR stsAborting;

// NETWORK 43
_w37 := stsStopped OR stsAborted OR stsPaused;
IF _w37 THEN stsMode := 0; END_IF
stsManual := _w37;

// NETWORK 44
_w38 := NOT stsManual;
IF _w38 THEN stsMode := 1; END_IF
stsAutomatic := _w38;

// NETWORK 45: Change Step Number to NextStep Reset the Step timer
_w39 := stsStep <> NextStep;
IF _w39 THEN stsStep := NextStep; END_IF
internalTimerReset S= _w39;

// NETWORK 46: Clear ActiveStep tag when transitioning to step 0.
R_TRIG_1(CLK := stsStep = 0); // R_TRIG
IF R_TRIG_1.Q THEN CurrentStep := internalClearStep; END_IF

// NETWORK 47: Step timer
_w40 := (NOT stsPaused OR stsPaused AND CompleteStateRequested) AND NOT internalTimerReset;
IF _w40 THEN StepTimer.PT := T#99H; END_IF
StepTimer(IN := _w40); // TON
stsStepTimerSeconds := TO_REAL(StepTimer.ET);
stsStepTimerSeconds := stsStepTimerSeconds / 1000;

// NETWORK 48
internalTimerReset R= internalTimerReset AND stsStep = NextStep;

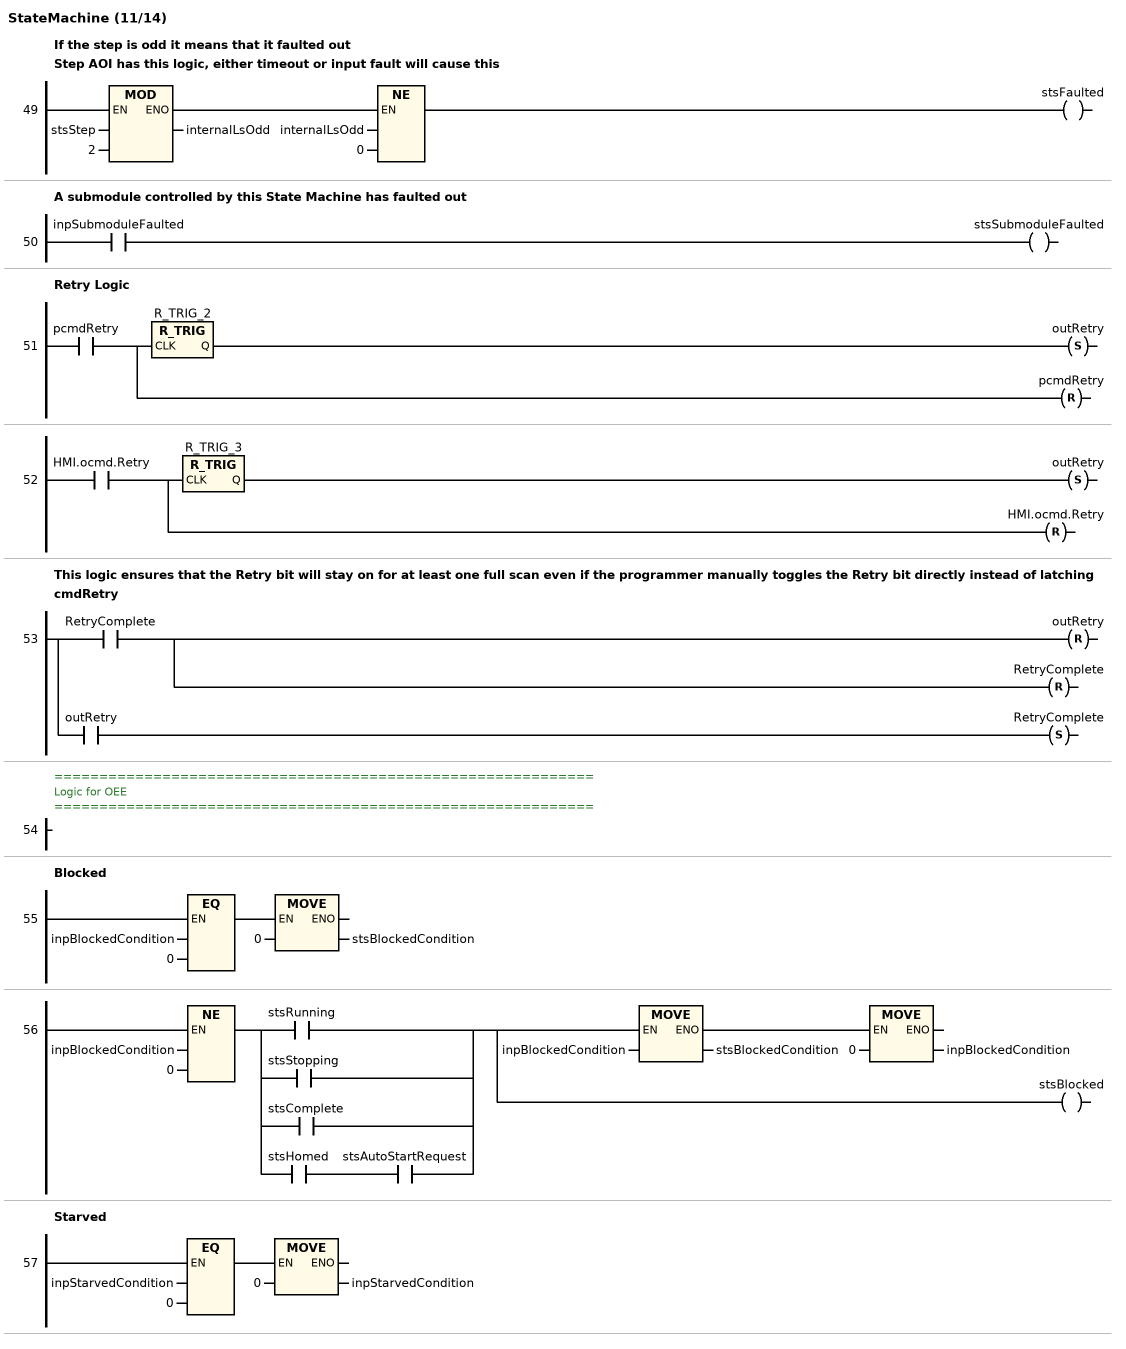
// NETWORK 49: If the step is odd it means that it faulted out Step AOI has this logic, either timeout or input fault will cause this
internalLsOdd := stsStep MOD 2;
stsFaulted := internalLsOdd <> 0;

// NETWORK 50: A submodule controlled by this State Machine has faulted out
stsSubmoduleFaulted := inpSubmoduleFaulted;

// NETWORK 51: Retry Logic
_w41 := pcmdRetry;
R_TRIG_2(CLK := _w41); // R_TRIG
outRetry S= R_TRIG_2.Q;
pcmdRetry R= _w41;

// NETWORK 52
_w42 := HMI.ocmd.Retry;
R_TRIG_3(CLK := _w42); // R_TRIG
outRetry S= R_TRIG_3.Q;
HMI.ocmd.Retry R= _w42;

// NETWORK 53: This logic ensures that the Retry bit will stay on for at least one full scan even if the programmer manually toggles the Retry bit directly instead of latching cmdRetry
outRetry R= RetryComplete;
RetryComplete R= RetryComplete;
RetryComplete S= outRetry;

// NETWORK 54
// ============================================================
// Logic for OEE
// ============================================================

// NETWORK 55: Blocked
IF inpBlockedCondition = 0 THEN stsBlockedCondition := 0; END_IF

// NETWORK 56
_w43 := inpBlockedCondition <> 0 AND (stsRunning OR stsStopping OR stsComplete OR stsHomed AND stsAutoStartRequest);
IF _w43 THEN stsBlockedCondition := inpBlockedCondition; END_IF
IF _w43 THEN inpBlockedCondition := 0; END_IF
stsBlocked := _w43;

// NETWORK 57: Starved
IF inpStarvedCondition = 0 THEN inpStarvedCondition := 0; END_IF

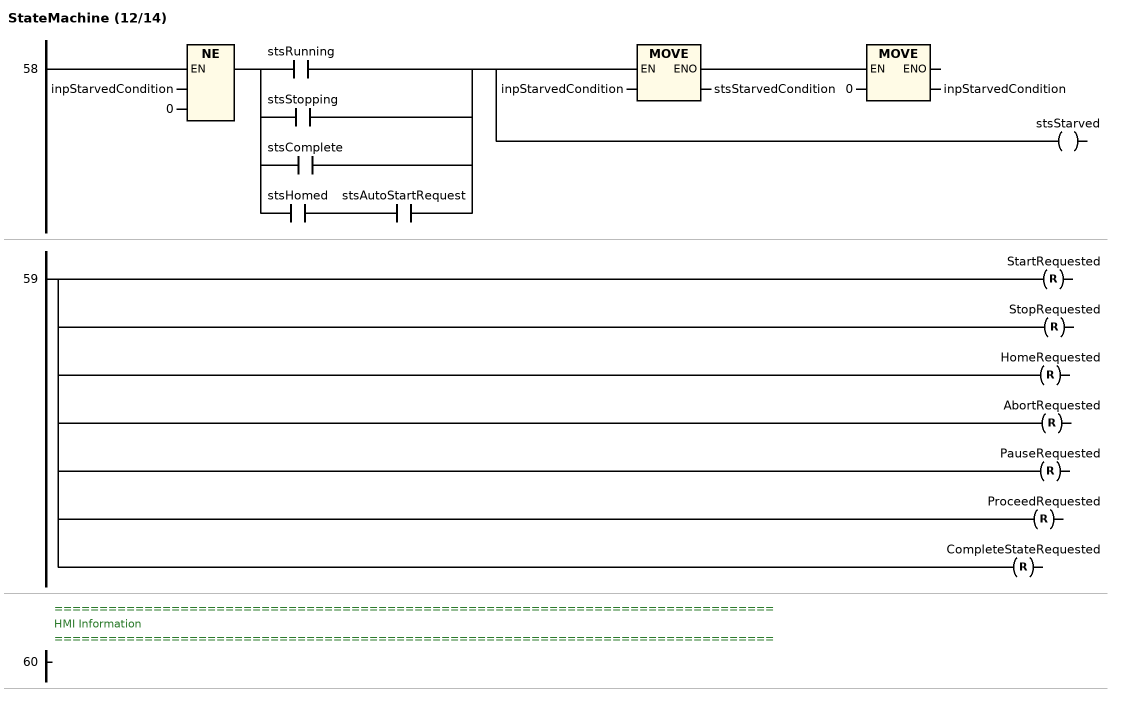
// NETWORK 58
_w44 := inpStarvedCondition <> 0 AND (stsRunning OR stsStopping OR stsComplete OR stsHomed AND stsAutoStartRequest);
IF _w44 THEN stsStarvedCondition := inpStarvedCondition; END_IF
IF _w44 THEN inpStarvedCondition := 0; END_IF
stsStarved := _w44;

// NETWORK 59
StartRequested R= TRUE;
StopRequested R= TRUE;
HomeRequested R= TRUE;
AbortRequested R= TRUE;
PauseRequested R= TRUE;
ProceedRequested R= TRUE;
CompleteStateRequested R= TRUE;

// NETWORK 60
// ================================================================================
//
// HMI Information
//
// ================================================================================

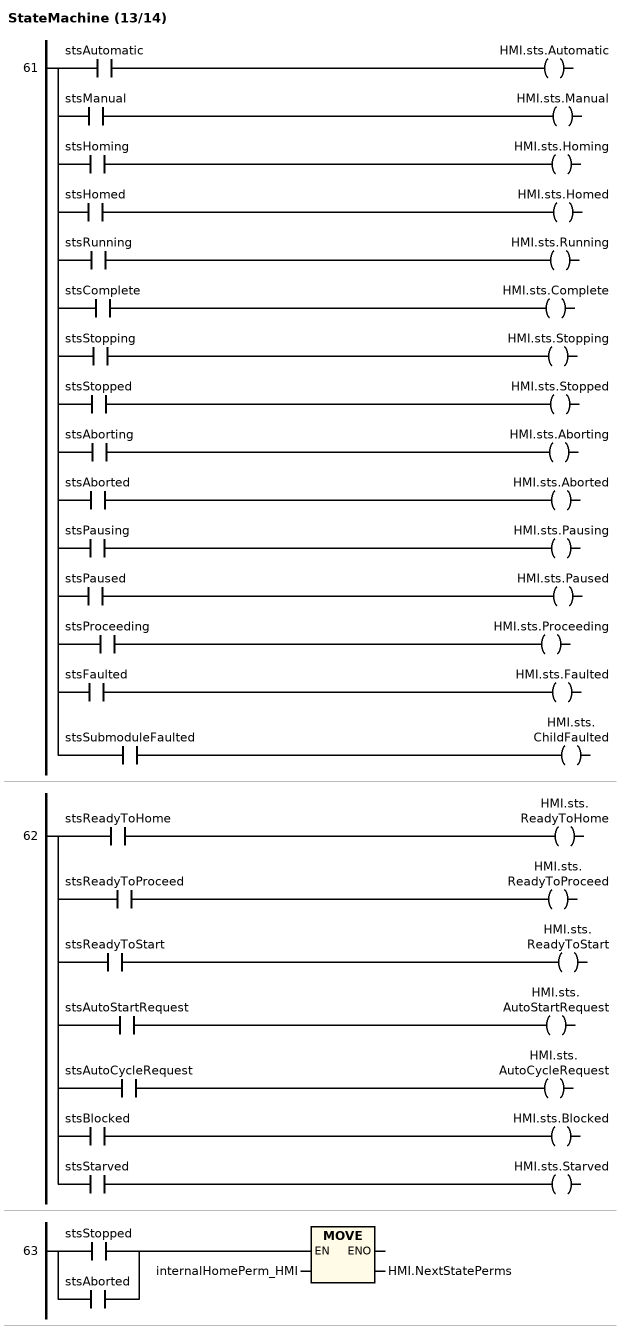
// NETWORK 61
HMI.sts.Automatic := stsAutomatic;
HMI.sts.Manual := stsManual;
HMI.sts.Homing := stsHoming;
HMI.sts.Homed := stsHomed;
HMI.sts.Running := stsRunning;
HMI.sts.Complete := stsComplete;
HMI.sts.Stopping := stsStopping;
HMI.sts.Stopped := stsStopped;
HMI.sts.Aborting := stsAborting;
HMI.sts.Aborted := stsAborted;
HMI.sts.Pausing := stsPausing;
HMI.sts.Paused := stsPaused;
HMI.sts.Proceeding := stsProceeding;
HMI.sts.Faulted := stsFaulted;
HMI.sts.ChildFaulted := stsSubmoduleFaulted;

// NETWORK 62
HMI.sts.ReadyToHome := stsReadyToHome;
HMI.sts.ReadyToProceed := stsReadyToProceed;
HMI.sts.ReadyToStart := stsReadyToStart;
HMI.sts.AutoStartRequest := stsAutoStartRequest;
HMI.sts.AutoCycleRequest := stsAutoCycleRequest;
HMI.sts.Blocked := stsBlocked;
HMI.sts.Starved := stsStarved;

// NETWORK 63
IF stsStopped OR stsAborted THEN HMI.NextStatePerms := internalHomePerm_HMI; END_IF

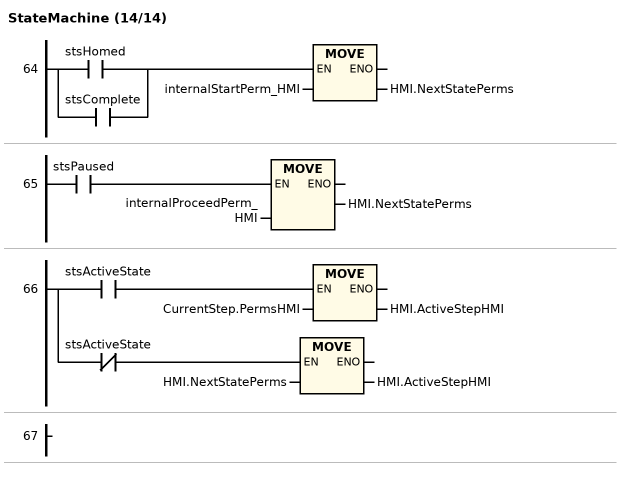
// NETWORK 64
IF stsHomed OR stsComplete THEN HMI.NextStatePerms := internalStartPerm_HMI; END_IF

// NETWORK 65
IF stsPaused THEN HMI.NextStatePerms := internalProceedPerm_HMI; END_IF

// NETWORK 66
IF stsActiveState THEN HMI.ActiveStepHMI := CurrentStep.PermsHMI; END_IF
IF NOT stsActiveState THEN HMI.ActiveStepHMI := HMI.NextStatePerms; END_IF

// NETWORK 67

END_FUNCTION_BLOCK

// Function Blocks/Step
FUNCTION_BLOCK Step
VAR_INPUT
	
	EN: BOOL;
	inpStep: DINT;
	cfgStep: DINT;
	cfgNextStep: DINT;
	cfgStepTimeOut: REAL;
	inpStepTimerSeconds: REAL;
	
	Permisives: INT := -1;
	inBypassPermissives: BOOL;
	inpFaultStep: BOOL;
	inpRetry: BOOL;
	
	
	
END_VAR
VAR_OUTPUT
	ENOut: BOOL;
	
	outStepActive: BOOL;
	outStepActiveOS: BOOL;
	outFaultedStepActive: BOOL;
	outFaultedStepActiveOS: BOOL;
	
	stsBypassed: BOOL;
	outActiveStepTimedOut: BOOL;
	
END_VAR
VAR
	
	
	R_TRIG_0: R_TRIG;
	R_TRIG_1: R_TRIG;
	R_TRIG_2: R_TRIG;
	
	internalHMI: PermIntlkHMI;
	Step_P_Perm: Permissives;
	
	
END_VAR


VAR_IN_OUT
	ActiveStep: ActiveStep;
	outNextStep: DINT;
END_VAR
VAR // added by the converter: edge detectors and wires of the graphical bodies
    _w1, _w2, _w3, _w4 : BOOL;
END_VAR

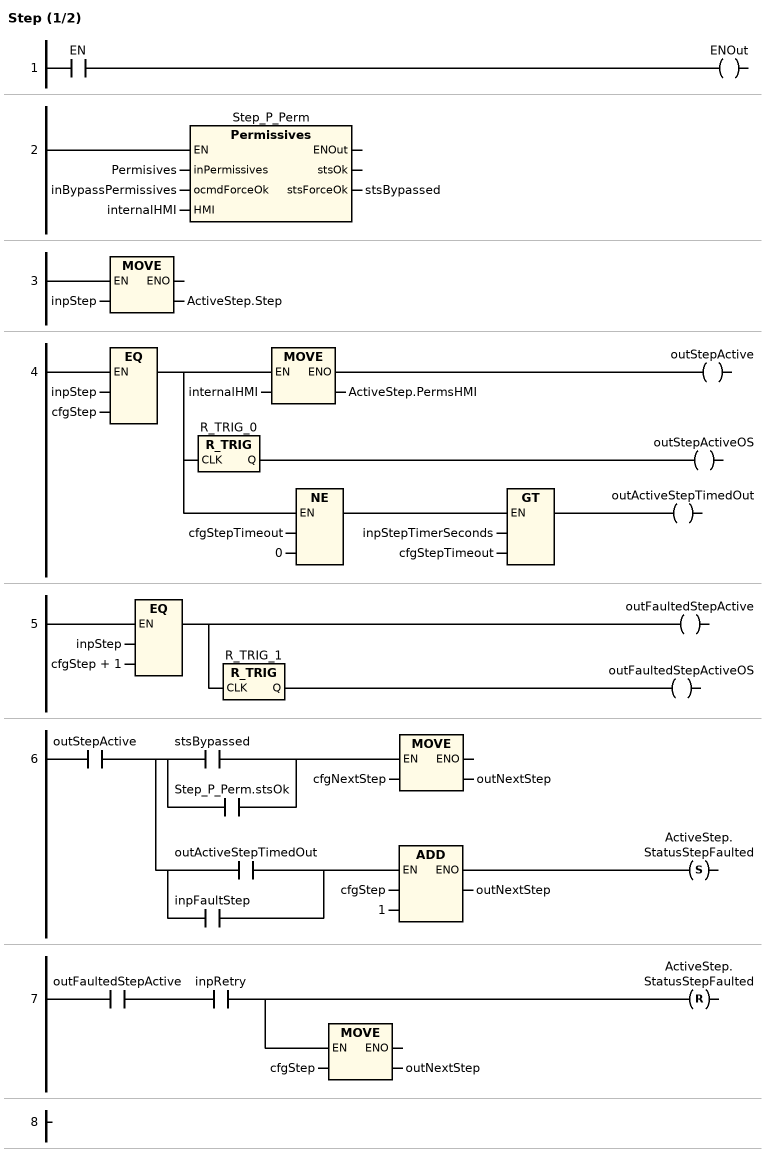
// NETWORK 1
ENOut := EN;

// NETWORK 2
Step_P_Perm(
    EN := TRUE,
    inPermissives := Permisives,
    ocmdForceOk := inBypassPermissives,
    HMI := internalHMI,
    stsForceOk => stsBypassed); // Permissives

// NETWORK 3
ActiveStep.Step := inpStep;

// NETWORK 4
_w1 := inpStep = cfgStep;
IF _w1 THEN ActiveStep.PermsHMI := internalHMI; END_IF
outStepActive := _w1;
R_TRIG_0(CLK := _w1); // R_TRIG
outStepActiveOS := R_TRIG_0.Q;
outActiveStepTimedOut := _w1 AND cfgStepTimeout <> 0 AND inpStepTimerSeconds > cfgStepTimeout;

// NETWORK 5
_w2 := inpStep = (cfgStep + 1);
outFaultedStepActive := _w2;
R_TRIG_1(CLK := _w2); // R_TRIG
outFaultedStepActiveOS := R_TRIG_1.Q;

// NETWORK 6
IF outStepActive AND (stsBypassed OR Step_P_Perm.stsOk) THEN outNextStep := cfgNextStep; END_IF
_w3 := outStepActive AND (outActiveStepTimedOut OR inpFaultStep);
IF _w3 THEN outNextStep := cfgStep + 1; END_IF
ActiveStep.StatusStepFaulted S= _w3;

// NETWORK 7
_w4 := outFaultedStepActive AND inpRetry;
ActiveStep.StatusStepFaulted R= _w4;
IF _w4 THEN outNextStep := cfgStep; END_IF

// NETWORK 8

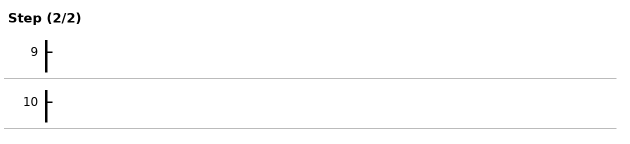
// NETWORK 9

// NETWORK 10

END_FUNCTION_BLOCK

// Visu_Logic/Visu_Logic
PROGRAM Visu_Logic
VAR
	permissivesOK : DINT;
	
END_VAR

// NETWORK 1

END_PROGRAM

// Visualizations/Button
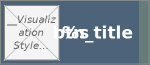
VISUALIZATION Button  // 150x65
VAR_INPUT
	
END_VAR

VAR 
	elemColor :DWORD := 16#FF314F60;
END_VAR
    Rectangle (-1,0 152x65), colour toggle: button_variable, colour variable: elemColor
        p3450524324: elemColor
        p3092690914: elemColor
        p2167032090: elemColor
        tap button_variable
        OnMouseClick: execute { elemColor := click_color; }
        OnMouseDown: execute { elemColor := mouseDown_color; }
        OnMouseEnter: execute { elemColor := hover_color; }
        OnMouseLeave: execute { elemColor := normal_color; }
    Rectangle (139,0 12x65), colour toggle: button_light, invisible if: hide_light, colour variable: led_colorOFF
        p3450524324: led_colorOFF
        p3092690914: led_colorON
        p2167032090: led_colorON
    Rectangle (15,19 121x27), "%s", text variable: button_text, invisible if: hide_text
    Image (4,5 55x55), invisible if: hide_image
        p84334746: button_image
    Rectangle (15,19 121x27), "btn_title", invisible if: hide_title
    Rectangle (-1,-1 152x65), colour toggle: button_variable, colour variable: elemColor
        p3450524324: elemColor
        p3092690914: elemColor
        p2167032090: elemColor
        tap button_variable
        OnMouseClick: execute { elemColor := click_color; }
        OnMouseDown: execute { elemColor := mouseDown_color; }
        OnMouseEnter: execute { elemColor := hover_color; }
        OnMouseLeave: execute { elemColor := normal_color; }
END_VISUALIZATION

// Visualizations/Menu_Button
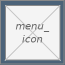
VISUALIZATION Menu_Button  // 65x65
VAR
	elemColor :DWORD := 16#FF314F60;
	button_variable : BOOL := FALSE;
	
END_VAR

VAR_IN_OUT
	deltaPos : INT := 0;
	invisibleTrue : BOOL;
END_VAR
    Rectangle (0,0 67x65), colour toggle: button_variable, colour variable: elemColor
        p3450524324: elemColor
        p3092690914: elemColor
        p2167032090: elemColor
        tap button_variable
        OnMouseLeave: execute { elemColor := normal_color; }
    Image (5,5 55x55), image: menu_icon
    Rectangle (0,0 67x65), colour toggle: button_variable, colour variable: elemColor
        p3450524324: elemColor
        p3092690914: elemColor
        p2167032090: elemColor
        tap button_variable
        OnMouseClick: execute { invisibleTrue := FALSE; elemColor := click_color; }
        OnMouseClick: execute {
            IF (deltaPos = -322) THEN
                deltaPos := 0;
            ELSIF (deltaPos = 0) THEN
                deltaPos := -322;
            END_IF;
        }
        OnMouseDown: execute { elemColor := mouseDown_color; }
        OnMouseEnter: execute { elemColor := hover_color; }
        OnMouseLeave: execute { elemColor := normal_color; }
END_VISUALIZATION

// Visualizations/Permissives_faceplate
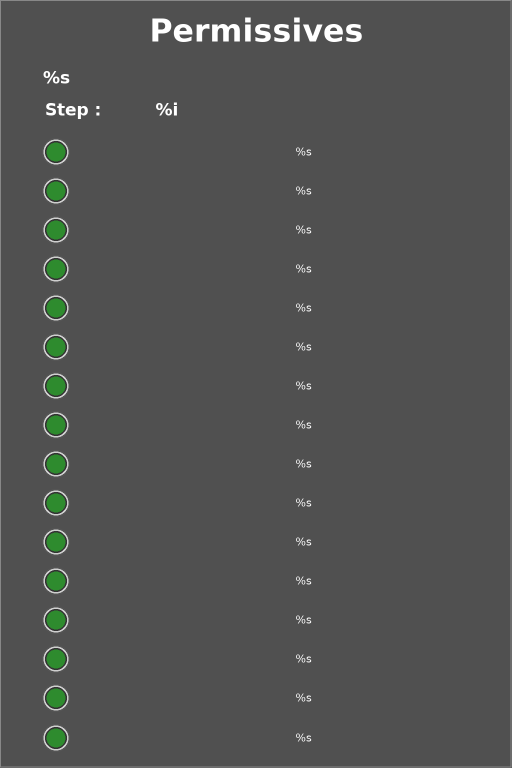
VISUALIZATION Permissives_faceplate  // 512x768
VAR_IN_OUT
	SM_Perm_Visualization_Tag : StateMachine;
END_VAR
    Label (125,-3 263x67), "Permissives"
    Group (40,136 429x32)
        Lamp1 (0,0 32x32), variable: SM_Perm_Visualization_Tag.CurrentStep.PermsHMI.sts.PermIntlk.0, style: Lamp-Lamp1-Green
        Textfield (98,0 331x32), "%s", text variable: SM_Perm_Visualization_Tag.HMI.ActiveStepHMI.cfg.Desc[0]
    Group (40,175 429x32)
        Lamp1 (0,0 32x32), variable: SM_Perm_Visualization_Tag.CurrentStep.PermsHMI.sts.PermIntlk.1, style: Lamp-Lamp1-Green
        Textfield (98,0 331x32), "%s", text variable: SM_Perm_Visualization_Tag.HMI.ActiveStepHMI.cfg.Desc[1]
    Group (40,214 429x32)
        Lamp1 (0,0 32x32), variable: SM_Perm_Visualization_Tag.CurrentStep.PermsHMI.sts.PermIntlk.2, style: Lamp-Lamp1-Green
        Textfield (98,0 331x32), "%s", text variable: SM_Perm_Visualization_Tag.HMI.ActiveStepHMI.cfg.Desc[2]
    Group (40,253 429x32)
        Lamp1 (0,0 32x32), variable: SM_Perm_Visualization_Tag.CurrentStep.PermsHMI.sts.PermIntlk.3, style: Lamp-Lamp1-Green
        Textfield (98,0 331x32), "%s", text variable: SM_Perm_Visualization_Tag.HMI.ActiveStepHMI.cfg.Desc[3]
    Group (40,292 429x32)
        Lamp1 (0,0 32x32), variable: SM_Perm_Visualization_Tag.CurrentStep.PermsHMI.sts.PermIntlk.4, style: Lamp-Lamp1-Green
        Textfield (98,0 331x32), "%s", text variable: SM_Perm_Visualization_Tag.HMI.ActiveStepHMI.cfg.Desc[4]
    Group (40,331 429x32)
        Lamp1 (0,0 32x32), variable: SM_Perm_Visualization_Tag.CurrentStep.PermsHMI.sts.PermIntlk.5, style: Lamp-Lamp1-Green
        Textfield (98,0 331x32), "%s", text variable: SM_Perm_Visualization_Tag.HMI.ActiveStepHMI.cfg.Desc[5]
    Group (40,370 429x32)
        Lamp1 (0,0 32x32), variable: SM_Perm_Visualization_Tag.CurrentStep.PermsHMI.sts.PermIntlk.6, style: Lamp-Lamp1-Green
        Textfield (98,0 331x32), "%s", text variable: SM_Perm_Visualization_Tag.HMI.ActiveStepHMI.cfg.Desc[6]
    Group (40,409 429x32)
        Lamp1 (0,0 32x32), variable: SM_Perm_Visualization_Tag.CurrentStep.PermsHMI.sts.PermIntlk.7, style: Lamp-Lamp1-Green
        Textfield (98,0 331x32), "%s", text variable: SM_Perm_Visualization_Tag.HMI.ActiveStepHMI.cfg.Desc[7]
    Group (40,448 429x32)
        Lamp1 (0,0 32x32), variable: SM_Perm_Visualization_Tag.CurrentStep.PermsHMI.sts.PermIntlk.8, style: Lamp-Lamp1-Green
        Textfield (98,0 331x32), "%s", text variable: SM_Perm_Visualization_Tag.HMI.ActiveStepHMI.cfg.Desc[8]
    Group (40,487 429x32)
        Lamp1 (0,0 32x32), variable: SM_Perm_Visualization_Tag.CurrentStep.PermsHMI.sts.PermIntlk.9, style: Lamp-Lamp1-Green
        Textfield (98,0 331x32), "%s", text variable: SM_Perm_Visualization_Tag.HMI.ActiveStepHMI.cfg.Desc[9]
    Group (40,526 429x32)
        Lamp1 (0,0 32x32), variable: SM_Perm_Visualization_Tag.CurrentStep.PermsHMI.sts.PermIntlk.10, style: Lamp-Lamp1-Green
        Textfield (98,0 331x32), "%s", text variable: SM_Perm_Visualization_Tag.HMI.ActiveStepHMI.cfg.Desc[10]
    Group (40,565 429x32)
        Lamp1 (0,0 32x32), variable: SM_Perm_Visualization_Tag.CurrentStep.PermsHMI.sts.PermIntlk.11, style: Lamp-Lamp1-Green
        Textfield (98,0 331x32), "%s", text variable: SM_Perm_Visualization_Tag.HMI.ActiveStepHMI.cfg.Desc[11]
    Group (40,604 429x32)
        Lamp1 (0,0 32x32), variable: SM_Perm_Visualization_Tag.CurrentStep.PermsHMI.sts.PermIntlk.12, style: Lamp-Lamp1-Green
        Textfield (98,0 331x32), "%s", text variable: SM_Perm_Visualization_Tag.HMI.ActiveStepHMI.cfg.Desc[12]
    Group (40,643 429x32)
        Lamp1 (0,0 32x32), variable: SM_Perm_Visualization_Tag.CurrentStep.PermsHMI.sts.PermIntlk.13, style: Lamp-Lamp1-Green
        Textfield (98,0 331x32), "%s", text variable: SM_Perm_Visualization_Tag.HMI.ActiveStepHMI.cfg.Desc[13]
    Group (40,682 429x32)
        Lamp1 (0,0 32x32), variable: SM_Perm_Visualization_Tag.CurrentStep.PermsHMI.sts.PermIntlk.14, style: Lamp-Lamp1-Green
        Textfield (98,0 331x32), "%s", text variable: SM_Perm_Visualization_Tag.HMI.ActiveStepHMI.cfg.Desc[14]
    Group (40,722 429x32)
        Lamp1 (0,0 32x32), variable: SM_Perm_Visualization_Tag.CurrentStep.PermsHMI.sts.PermIntlk.15, style: Lamp-Lamp1-Green
        Textfield (98,0 331x32), "%s", text variable: SM_Perm_Visualization_Tag.HMI.ActiveStepHMI.cfg.Desc[15]
    Rectangle (2,113 502x1022)
        OnMouseClick:  Dialog=Current Dialog, Result=OK, NumpadKeypadSet=True
    Textfield (40,69 429x17), "%s", text variable: SM_Perm_Visualization_Tag.HMI.ActiveStepHMI.cfg.Name
    Textfield (42,101 429x17), "Step : %i", text variable: SM_Perm_Visualization_Tag.stsStep
END_VISUALIZATION

// Visualizations/Screen_Navigation
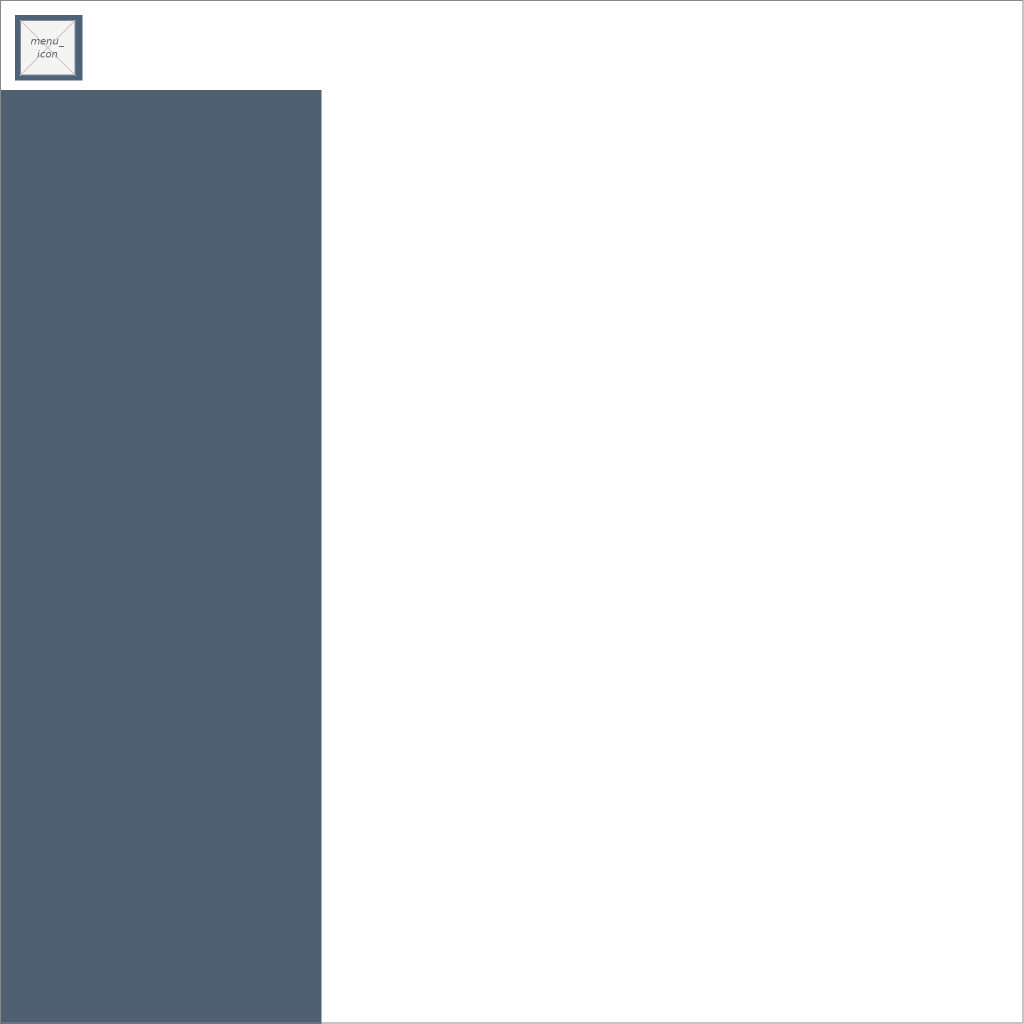
VISUALIZATION Screen_Navigation  // 1024x1024
VAR
	menuPos : Int := -322;
	hideMenu : BOOL := TRUE;
END_VAR
    Rectangle (-1,90 322x934)
        p3560616238: menuPos
    Frame (15,15 65x65)
        shows Menu_Button(menu_move := menuPos, invisibleTrue := hideMenu)
END_VISUALIZATION

// Visualizations/SM_faceplate
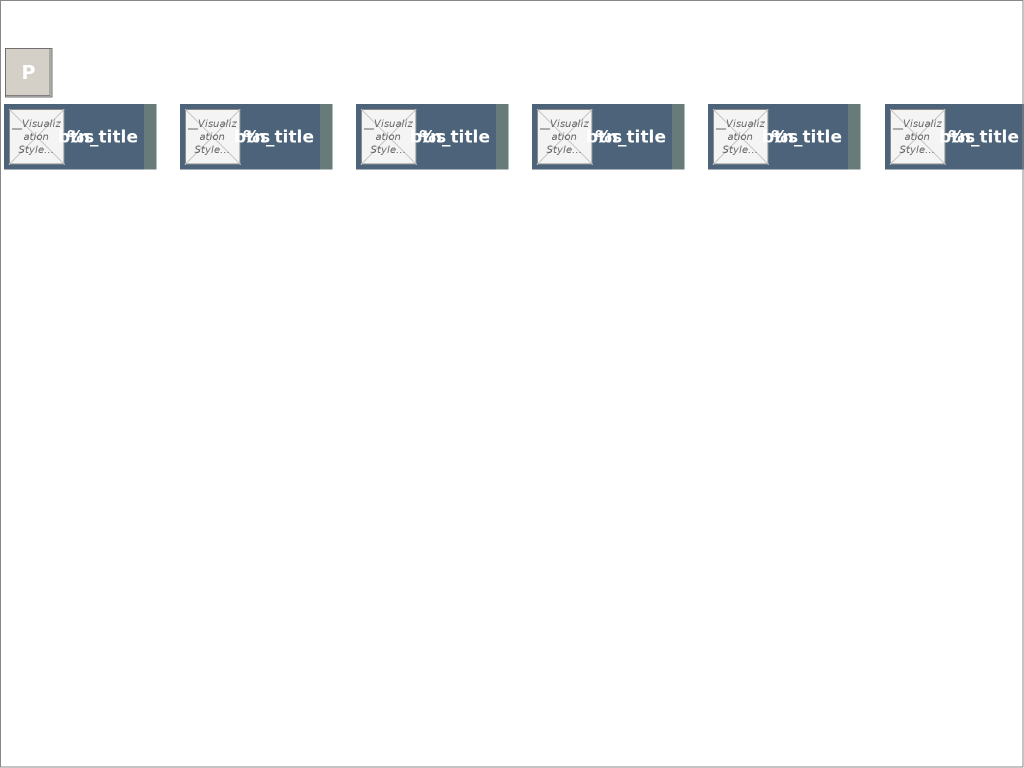
VISUALIZATION SM_faceplate  // 1024x768
VAR_IN_OUT
    SM_Visualization_Tag : StateMachine;
END_VAR

VAR
    // Dark Theme Colors for Visualization
    indicatorRed: DWORD := 16#FF800000;      // Standard red color, fully opaque
    indicatorGreen: DWORD := 16#FF008000;    // Standard green color, fully opaque

    // Modern Dark Color Palette for Buttons
    buttonRed: DWORD := 16#FFC21807;         // Dark rosy red, opaque
    buttonRedDarker1: DWORD := 16#FF911205;  // Crimson Red, opaque
    buttonRedDarker2: DWORD := 16#FF610C03;  // Dark Red, opaque
    buttonRedDarkest: DWORD := 16#FF300601;  // Maroon, opaque
    
    buttonGreen: DWORD := 16#FF0A7E07;       // Dark light green, opaque
    buttonGreenDarker1: DWORD := 16#FF075E05; // Medium Sea Green, opaque
    buttonGreenDarker2: DWORD := 16#FF053F03; // Dark Green, opaque
    buttonGreenDarkest: DWORD := 16#FF021F01; // Dark Olive Green, opaque
    
    buttonGrey: DWORD := 16#FF606060;        // Dark blue grey, opaque
    buttonGreyDarker1: DWORD := 16#FF484848; // Cadet Blue, opaque
    buttonGreyDarker2: DWORD := 16#FF303030; // Steel Blue, opaque
    buttonGreyDarkest: DWORD := 16#FF181818; // Dark Slate Gray, opaque

    buttonBlue: DWORD := 16#FF0D47A1;        // Modern Blue, opaque
    buttonBlueDarker1: DWORD := 16#FF093578; // Darker Blue, opaque
    buttonBlueDarker2: DWORD := 16#FF062350; // Even Darker Blue, opaque
    buttonBlueDarkest: DWORD := 16#FF031128; // Darkest Blue, opaque
    
    buttonPurple: DWORD := 16#FF6A1B9A;      // Modern Purple, opaque
    buttonPurpleDarker1: DWORD := 16#FF4F1473;// Darker Purple, opaque
    buttonPurpleDarker2: DWORD := 16#FF350D4D;// Even Darker Purple, opaque
    buttonPurpleDarkest: DWORD := 16#FF1A0626;// Darkest Purple, opaque

    buttonOrange: DWORD := 16#FFE65100;      // Modern Orange, opaque
    buttonOrangeDarker1: DWORD := 16#FFAC3C00;// Darker Orange, opaque
    buttonOrangeDarker2: DWORD := 16#FF732800;// Even Darker Orange, opaque
    buttonOrangeDarkest: DWORD := 16#FF391400;// Darkest Orange, opaque

    buttonYellow: DWORD := 16#FFFBC02D;      // Modern Yellow, opaque
    buttonYellowDarker1: DWORD := 16#FFBC9021;// Darker Yellow, opaque
    buttonYellowDarker2: DWORD := 16#FF7D6016;// Even Darker Yellow, opaque
    buttonYellowDarkest: DWORD := 16#FF3E300B;// Darkest Yellow, opaque
END_VAR
    Label (1,3 243x35), "State Machine"
    Textfield (63,48 225x22), "Step : %i", text variable: SM_Visualization_Tag.stsStep
    Textfield (351,48 225x22), "State : %s", text variable: SM_Visualization_Tag.stsStateString
    Textfield (62,75 225x22), "Step Timer : %i s", text variable: SM_Visualization_Tag.stsStepTimerSeconds
    Button (5,48 47x49), "P"
        p2175578022: buttonGreyDarker2
        OnMouseClick:  Dialog=Permissives_faceplate, Parameters={SM_Perm_Visualization_Tag: SM_Visualization_Tag}, OpenModal=True, OpenCentered=True, PositionX=-30, PositionY=-15
    Textfield (351,75 225x22), "Next State : %s", text variable: SM_Visualization_Tag.HMI.NextStatePerms.cfg.Name
    Frame (5,104 150x65)
        shows Button(Title := Abort, Hide_Title := False, Hide_Text := True, Image := 'ImagePool.abort_symbol', Hide_Image := False, Hide_Light := True, Button_Variable := SM_Visualization_Tag.pcmdAbort)
    Frame (181,104 150x65)
        shows Button(Title := Home, Hide_Title := False, Hide_Text := True, Image := 'ImagePool.home_symbol', Hide_Image := False, Button_Light := SM_Visualization_Tag.stsReadyToHome, Hide_Light := False, Button_Variable := SM_Visualization_Tag.pcmdHome)
    Frame (357,104 150x65)
        shows Button(Title := Start, Hide_Title := False, Hide_Text := True, Image := 'ImagePool.start_symbol', Hide_Image := False, Button_Light := SM_Visualization_Tag.stsReadyToStart, Hide_Light := False, Button_Variable := SM_Visualization_Tag.pcmdStart)
    Frame (533,104 150x65)
        shows Button(Title := Pause, Hide_Title := False, Hide_Text := True, Image := 'ImagePool.pause_symbol', Hide_Image := False, Hide_Light := True, Button_Variable := SM_Visualization_Tag.pcmdPause)
    Frame (709,104 150x65)
        shows Button(Title := Proceed, Hide_Title := False, Hide_Text := True, Image := 'ImagePool.proceed_symbol', Hide_Image := False, Button_Light := SM_Visualization_Tag.stsReadyToProceed, Hide_Light := False, Button_Variable := SM_Visualization_Tag.pcmdProceed)
    Frame (886,104 150x65)
        shows Button(Title := Retry, Hide_Title := False, Hide_Text := True, Image := 'ImagePool.retry_symbol', Hide_Image := False, Hide_Light := True, Button_Variable := SM_Visualization_Tag.pcmdRetry)
END_VISUALIZATION
